(*!
<summary>Advances the cursor to the next source position.</summary>
<description>
The source must be live, non-null and structurally unchanged during traversal. TRUE identifies a current
entry. The index advances only while below source Length and stops at the end position. Repeated exhausted
calls return FALSE without incrementing the index; reading Current yields an empty descriptor. Reset allows
traversal from the beginning again. No snapshot or mutation detection is provided. Descendants cannot override
this cursor operation; advancement, reset and borrowed current views use the same cursor state.
Missing source raises DataMemberNotSpecifiedException before source access or cursor advancement.
</description>
*)
{attribute "object_name" := "MoveNext"}
METHOD FINAL MoveNext : BOOL
requireSource();

IF _CurrentIndex < _List.Length THEN
	_CurrentIndex := _CurrentIndex + 1;
END_IF

MoveNext := _CurrentIndex < _List.Length;
END_METHOD

(*!
<summary>Provides the library namespace for diagnostics.</summary>
<description>
Borrowed read-only reference to compiler-initialized metadata; no ownership transfer.
</description>
*)
{attribute 'monitoring' := 'call'}
PROPERTY NamespaceName : REFERENCE TO STRING
GET
NamespaceName REF= CurrentNamespace.Name;
END_GET
END_PROPERTY

(*!
<summary>Places the cursor before the first source entry.</summary>
<description>
The next MoveNext starts at zero. Does not modify the source or release payload; reading Current now yields an
empty descriptor. Descendants cannot override this cursor operation; advancement, reset and borrowed current
views use the same cursor state.
</description>
*)
{attribute "object_name" := "Reset"}
METHOD FINAL Reset
_CurrentIndex := -1;
END_METHOD

(*!
<summary>Reports the size of this function-block instance.</summary>
<description>
Measured in bytes; includes inline storage but excludes separately allocated buffers, payload and enumerators.
</description>
*)
{attribute 'monitoring' := 'call'}
PROPERTY SelfSize : ULINT
GET
SelfSize := XSIZEOF(THIS^);
END_GET
END_PROPERTY

(*!
<summary>Requires the configured source before traversal or current-value access.</summary>
<description>
A missing mandatory source is configuration failure, not an empty collection. Raises a framework diagnostic
outside lifecycle methods and before mutation; it does not validate arbitrary pointer lifetime.
</description>
*)
METHOD PRIVATE requireSource
IF _List = 0 THEN
	TOF_Core.Exceptions.ThrowDataMemberNotSpecified(
		sourceNamespaceName := NamespaceName,
		sourceClassName := ClassName,
		sourcePOUName := __POUNAME(),
		sourcePosition := __POSITION(),
		dataMemberName := 'list'
	);
END_IF
END_METHOD

END_FUNCTION_BLOCK

// ---- List/List.TcPOU
(*
SPDX-FileCopyrightText: © 2026 Oleksandr Tiutyk <trofimich@gmail.com>
SPDX-License-Identifier: MIT
License: https://opensource.org/license/mit
*)

(*!
<summary>Stores an ordered sequence of generic values with fixed or dynamic capacity.</summary>
<description>
CreateEnumerator allocates an independent cursor owned by its caller. The collection must remain alive while
that cursor is used. Dynamic growth preserves the existing buffer on allocation failure and invokes the
terminal allocation-failure mechanism. Sort uses GENERIC_VALUE.CompareTo unless an explicit borrowed comparer
is supplied; descriptors preserve OBJECT and USER_DEFINED categories. Successful insertion transfers disposal
responsibility for owned payload; borrowed payload must remain alive while stored. The caller-side descriptor
copy is not reset and must not be released again after transfer. Independent owning aliases and overlapping
owned allocations are unsupported. Entries retain order and duplicates. Same-allocation replacement preserves
ownership without releasing retained storage. Get, FindSingle and enumerators only borrow payload.
ContainsGeneric defaults to releasing its query. Validators are borrowed for the collection lifetime. No
locking or mutation-version checks are implemented; callbacks that mutate the collection can invalidate
in-progress operations. Generic lookup with requested query release also attempts cleanup on lookup failure
before propagating the captured exception; terminal OOM takes precedence.
Instances cannot be assigned by value: copying backing pointers or disposal responsibility would create
unsafe aliases. Interface references still borrow this instance; copying an interface does not clone storage.
</description>
*)

{attribute 'no_explicit_call' := 'do not call this function block directly'}
FUNCTION_BLOCK List 
VAR_GENERIC CONSTANT
 	{attribute 'hide'} 
	//! <summary>Inline capacity; zero selects dynamic backing storage.</summary>
	_StaticCapacity : TOF_Core.DINT_LENGTH := 0;
END_VAR
EXTENDS TOF_Core.Object IMPLEMENTS IList
VAR_INPUT
	//! <summary>Number of slots added when dynamic storage is full; must be positive when growth is required.</summary>
	DefaultDynamicAllocationElementCount : BYTE := 10;	
END_VAR
VAR_STAT
	//! <summary>Class name shared by all instances of this function block.</summary>
	{attribute 'hide'} 
	_ClassName : STRING := __POUNAME();
END_VAR
VAR
	{attribute 'hide'} 
	_ValueValidator : TOF_Core.IGenericValueValidator;

	{attribute 'hide'} 
	_Array : POINTER TO TOF_Core.GENERIC_VALUE;
	{attribute 'hide'} 
	_StaticArray : ARRAY [0.._StaticCapacity - 1] OF TOF_Core.GENERIC_VALUE;
	
	{attribute 'hide'} 
	_DynamicCapacity : TOF_Core.DINT_LENGTH;
	{attribute 'hide'} 
	_Length : TOF_Core.DINT_LENGTH;
END_VAR

(*!
<summary>Grows the dynamic element buffer while preserving existing values.</summary>
<description>
Static instances return without allocation. A positive increment must fit DINT capacity and the UDINT
allocation-byte limit; invalid ranges raise ArgumentOutOfRangeException before storage changes. A null
allocation invokes the terminal allocation-failure mechanism before copying or deleting the old buffer.
Existing descriptors are moved without cloning payload; incoming ownership is not accepted by this helper.
Descendants cannot override this storage operation; capacity, indexing and disposal remain governed by this
collection implementation.
</description>
*)
METHOD PROTECTED FINAL AllocateMemory 
VAR_INPUT
	elementCount : TOF_Core.DINT_LENGTH;
END_VAR
VAR CONSTANT
	//! <summary>Bytes per capacity slot, including descriptor storage and any hash-index arrays.</summary>
	ENTRY_ALLOCATION_SIZE : ULINT := XSIZEOF(TOF_Core.GENERIC_VALUE);
END_VAR
VAR
	newMemory : POINTER TO TOF_Core.GENERIC_VALUE;
	newCapacity : ULINT;

END_VAR
IF NOT Dynamic THEN
	RETURN;
END_IF

IF elementCount <= TOF_Core.SignedInt32.ZERO THEN
	TOF_Core.Exceptions.ThrowArgumentOutOfRange(
		sourceNamespaceName := NamespaceName,
		sourceClassName := ClassName,
		sourcePOUName := __POUNAME(),
		sourcePosition := __POSITION(),
		argumentName := 'elementCount',
		argumentValue := elementCount
	);
END_IF

newCapacity := TO_ULINT(_DynamicCapacity) + TO_ULINT(elementCount);

IF newCapacity > TO_ULINT(TOF_Core.SignedInt32.MAX_VALUE)
	OR_ELSE newCapacity > TO_ULINT(TOF_Core.UnsignedInt32.MAX_VALUE) / ENTRY_ALLOCATION_SIZE
THEN
	TOF_Core.Exceptions.ThrowArgumentOutOfRange(
		sourceNamespaceName := NamespaceName,
		sourceClassName := ClassName,
		sourcePOUName := __POUNAME(),
		sourcePosition := __POSITION(),
		argumentName := 'capacity',
		argumentValue := newCapacity
	);
END_IF

newMemory := __NEW(BYTE, TO_UDINT(ENTRY_ALLOCATION_SIZE * newCapacity));

IF newMemory = 0 THEN
	TOF_Core.DynamicMemoryManager.RaiseAllocationFailure();
END_IF

IF _Length > TOF_Core.SignedInt32.ZERO THEN
	Tc2_System.MEMCPY(destAddr := newMemory, srcAddr := _Array, n := TO_UDINT(ENTRY_ALLOCATION_SIZE * TO_ULINT(_Length)));
END_IF

IF _Array <> 0 THEN
	__DELETE(_Array);
END_IF

_DynamicCapacity := TO_DINT(newCapacity);
_Array := newMemory;
END_METHOD

(*!
<summary>Copies a value and appends the owned descriptor.</summary>
<description>
Borrows the original during the call. isObject = TRUE requires a live Object FB instance implementing
ICloneable; other data is copied as bytes without recursively cloning references. A prepared copy is released
if insertion fails before acceptance; exceptions propagate. Engine-managed exception objects are unsupported.
index is meaningful only on success. Descendants cannot override this storage operation; capacity, indexing
and disposal remain governed by this collection implementation.
The original failure is captured before cleanup so nested cleanup handling cannot replace its payload.
A static native wrapper is cloned before cleanup; failure to capture still attempts prepared-copy disposal.
Terminal allocation failure takes precedence and no exception clone is allocated after its latch is set.
</description>
*)
METHOD FINAL AppendCopy : IList
VAR_INPUT
	value : ANY;
	isObject : BOOL := FALSE;
END_VAR
VAR_OUTPUT
	index : TOF_Core.DINT_INDEX;
END_VAR
VAR
	exceptionCode : __SYSTEM.ExceptionCode;
	caughtException : TOF_Core.IException;
	genericValue : TOF_Core.GENERIC_VALUE;
END_VAR

genericValue := TOF_Core.GenericValueFactory.FromAnyType(
		value := value,
		isObject := isObject,
		memoryManagementBehavior := TOF_Core.GENERIC_MEMORY_MANAGEMENT_BEHAVIOR.CLONE_ORIGINAL_VALUE_AND_OWNS_MEMORY
	);

__TRY
	AppendCopy := AppendGeneric(value := genericValue, index => index);
__CATCH(exceptionCode)
	caughtException := TOF_Core.ExceptionManager.GetLastException(
		exceptionCode := exceptionCode,
		catchPointNamespaceName := NamespaceName,
		catchPointPOUName := __POUNAME(),
		catchPointPosition := __POSITION()
	);
__ENDTRY

IF caughtException <> 0 THEN
	__TRY
		TOF_Core.DynamicMemoryManager.RaiseIfAllocationFailed();

		IF NOT caughtException.IsDynamicInstance THEN
			__QUERYINTERFACE(caughtException.Clone(), caughtException);
		END_IF
	__CATCH(exceptionCode)
		genericValue.Release();

		TOF_Core.ExceptionManager.ReThrowLastException(
			exceptionCode := exceptionCode,
			catchPointNamespaceName := NamespaceName,
			catchPointPOUName := __POUNAME(),
			catchPointPosition := __POSITION()
		);
	__ENDTRY

	genericValue.Release();

	TOF_Core.ExceptionManager.Throw(exception := caughtException);
END_IF
END_METHOD

(*!
<summary>Appends a descriptor to the list.</summary>
<description>
Successful insertion transfers disposal responsibility for owned payload; borrowed payload must remain alive
while stored. The caller-side descriptor copy is not reset and must not be released again after transfer.
Independent owning aliases and overlapping owned allocations are unsupported. Delegates to InsertGeneric;
index is meaningful only on success. Descendants cannot override this storage operation; capacity, indexing
and disposal remain governed by this collection implementation.
</description>
*)
METHOD FINAL AppendGeneric : IList
VAR_INPUT
	value : TOF_Core.GENERIC_VALUE;
END_VAR
VAR_OUTPUT
	index : TOF_Core.DINT_INDEX;
END_VAR
index := _Length;

AppendGeneric := InsertGeneric(index := index, value := value);
END_METHOD

(*!
<summary>Reports the currently allocated number of slots.</summary>
<description>
Units are bytes for ByteList and entries for other collections. Static capacity is fixed; dynamic capacity can
change on growth or clearing. This is not a guarantee that the next allocation succeeds.
</description>
*)
{attribute 'monitoring' := 'call'}
PROPERTY FINAL Capacity : TOF_Core.DINT_LENGTH
GET
Capacity := SEL(_StaticCapacity = 0, _StaticCapacity, _DynamicCapacity);
END_GET
END_PROPERTY

(*!
<summary>Borrows the concrete collection class name without transferring storage ownership.</summary>
*)
{attribute 'monitoring' := 'call'}
PROPERTY ClassName : REFERENCE TO STRING
GET
ClassName REF= _ClassName;
END_GET
END_PROPERTY

(*!
<summary>Removes all entries and releases dynamic backing storage.</summary>
<description>
Owned payload is released best effort through GENERIC_VALUE.Release; borrowed storage is not freed. Static
capacity and the borrowed validator are retained. Dynamic capacity becomes zero. Returns this collection and
invalidates positions and views. Cleanup callbacks must not reenter mutation. Descendants cannot override this
storage operation; capacity, indexing and disposal remain governed by this collection implementation.
</description>
*)
METHOD FINAL Clear : IList
VAR
	i : DINT;
END_VAR
Clear := THIS^;

FOR i := 0 TO _Length - 1 DO
	_Array[i].Release();						
END_FOR	

_Length := 0;
_DynamicCapacity := 0;

IF _Array <> 0 AND_THEN Dynamic THEN
	__DELETE(_Array);	
END_IF
END_METHOD

(*!
<summary>Searches for a value using default generic equality.</summary>
<description>
Borrows the ANY argument during a linear search without cloning or releasing it. isObject = TRUE means a live
Object FB instance, not a pointer or interface variable. Equality exceptions propagate; callbacks that mutate
the collection can invalidate traversal. Descendants cannot override this storage operation; capacity,
indexing and disposal remain governed by this collection implementation.
</description>
*)
METHOD FINAL Contains : BOOL
VAR_INPUT
	value : ANY;
	isObject : BOOL := FALSE;
END_VAR
VAR
	genericValue : TOF_Core.GENERIC_VALUE;
	i : TOF_Core.DINT_INDEX;
END_VAR

genericValue := TOF_Core.GenericValueFactory.FromAnyType(
		value := value,
		isObject := isObject,
		memoryManagementBehavior := TOF_Core.GENERIC_MEMORY_MANAGEMENT_BEHAVIOR.STORE_ORIGINAL_REFERENCE_AND_NOT_OWNS_MEMORY
	);

FOR i := 0 TO _Length - 1 DO
	IF _Array[i].Equals(otherValue := genericValue) THEN
		Contains := TRUE;
		RETURN;
	END_IF
END_FOR
END_METHOD

(*!
<summary>Searches for an equal generic value and optionally releases the query.</summary>
<description>
Uses GENERIC_VALUE.Equals in a linear search. releaseValue defaults to TRUE: after a completed search, Release
is called on the local query copy, including on a miss. Caller-side aliases are not reset. The query must not
own storage retained by the collection. Requested release is attempted after both successful lookup and lookup
failure. Before cleanup, the original framework exception is retained and a borrowed static system exception
is cloned to preserve its code, catch point and timestamps across cleanup callbacks. The captured exception is
then propagated through ExceptionManager.Throw in the current cyclic task; native errors use the framework
SystemException representation. If capturing the system exception fails with terminal OOM, query cleanup is
still attempted and terminal OOM takes precedence. Terminal allocation state is never cleared. Release is best
effort and does not prove successful deallocation. Cleanup callbacks must not reenter collection mutation.
Descendants cannot override this storage operation; capacity, indexing and disposal remain governed by this
collection implementation.
</description>
*)
METHOD FINAL ContainsGeneric : BOOL
VAR_INPUT
	value : TOF_Core.GENERIC_VALUE;
	releaseValue : BOOL := TRUE;
END_VAR
VAR
	exceptionCode : __SYSTEM.ExceptionCode;
	caughtException : TOF_Core.IException;

	i : DINT;
END_VAR
__TRY
	FOR i := 0 TO _Length - 1 DO
		IF _Array[i].Equals(otherValue := value) THEN
			ContainsGeneric := TRUE;
			EXIT;
		END_IF
	END_FOR
__CATCH(exceptionCode)
	caughtException := TOF_Core.ExceptionManager.GetLastException(
		exceptionCode := exceptionCode,
		catchPointNamespaceName := NamespaceName,
		catchPointPOUName := __POUNAME(),
		catchPointPosition := __POSITION()
	);
__ENDTRY

IF releaseValue THEN
	IF caughtException <> 0 AND_THEN NOT caughtException.IsDynamicInstance THEN
		__TRY
			TOF_Core.DynamicMemoryManager.RaiseIfAllocationFailed();
			__QUERYINTERFACE(caughtException.Clone(), caughtException);
		__CATCH(exceptionCode)
			value.Release();

			TOF_Core.ExceptionManager.ReThrowLastException(
				exceptionCode := exceptionCode,
				catchPointNamespaceName := NamespaceName,
				catchPointPOUName := __POUNAME(),
				catchPointPosition := __POSITION()
			);
		__ENDTRY
	END_IF

	value.Release();
END_IF

IF caughtException <> 0 THEN
	TOF_Core.ExceptionManager.Throw(exception := caughtException);
END_IF
END_METHOD

(*!
<summary>Creates an independent enumerator owned by the caller.</summary>
<description>
The caller must explicitly release the enumerator and keep this collection alive while using it. Allocation
failure invokes DynamicMemoryManager.RaiseAllocationFailure without a heap exception; it is terminal and is
not returned as a recoverable null result.
</description>
*)
METHOD CreateEnumerator : TOF_Core.IEnumerator
VAR
	enumerator : POINTER TO ListEnumerator;
END_VAR
enumerator := __NEW(ListEnumerator(list := THIS^));

IF enumerator = 0 THEN
	TOF_Core.DynamicMemoryManager.RaiseAllocationFailure();
END_IF

CreateEnumerator := enumerator^;
END_METHOD

(*!
<summary>Reports whether storage can grow dynamically.</summary>
<description>
Static capacity zero selects dynamic storage. Dynamic collections can still fail to allocate.
</description>
*)
{attribute 'monitoring' := 'call'}
PROPERTY FINAL Dynamic : BOOL
GET
Dynamic := _StaticCapacity = 0;
END_GET
END_PROPERTY

(*!
<summary>Reports whether the collection has no entries.</summary>
<description>
Reflects Length; not a check of payload lifetime or memory health.
</description>
*)
{attribute 'monitoring' := 'call'}
PROPERTY FINAL Empty : BOOL
GET
Empty := _Length <= 0;
END_GET
END_PROPERTY

(*!
<summary>Releases owned payload and backing storage during destruction.</summary>
<description>
Calls Clear; lifecycle methods and payload cleanup callbacks must not raise exceptions or reenter mutation.
Payload release is best effort, not proof of successful destruction. No separate copy-code ownership handoff
is implemented.
</description>
*)

METHOD FB_exit : BOOL
VAR_INPUT
	bInCopyCode : BOOL; 
END_VAR
Clear();
END_METHOD

(*!
<summary>Binds the optional validator and inline storage during initialization.</summary>
<description>
The validator is borrowed and must remain alive while used; it is not invoked here. Static storage is bound
without allocation. Lifecycle methods must not raise exceptions. No explicit online-change relocation repair
is implemented.
</description>
*)
METHOD FB_init : BOOL
VAR_INPUT
	bInitRetains : BOOL; // TRUE: the retain variables are initialized (reset warm / reset cold)
	bInCopyCode : BOOL; // TRUE: the instance will be copied to the copy code afterward (online change)
	valueValidator : TOF_Core.IGenericValueValidator;
END_VAR
_ValueValidator := valueValidator;

IF NOT Dynamic THEN
	_Array := ADR(_StaticArray); 
END_IF
END_METHOD

(*!
<summary>Finds a predicate match in the requested traversal direction.</summary>
<description>
skip counts matches, not visited entries. A null predicate or no match returns FALSE; outputs are meaningful
only on TRUE. The result is borrowed even if IsMemoryOwner is TRUE. Predicate input uses AsAnyType without
preserving the explicit generic OBJECT category. Predicate exceptions propagate; callbacks must not mutate the
traversed collection. Descendants cannot override this storage operation; capacity, indexing and disposal
remain governed by this collection implementation.
</description>
*)
METHOD FINAL FindSingle : BOOL
VAR_INPUT
	predicate : TOF_Core.IPredicate;
	skip : UDINT := 0;
	searchDirection : TOF_Core.SEARCH_DIRECTION := TOF_Core.SEARCH_DIRECTION.FROM_BEGINNING;
END_VAR
VAR_OUTPUT
	value : TOF_Core.GENERIC_VALUE;
	index : TOF_Core.DINT_INDEX;
END_VAR
VAR
	startSearchIndex : DINT;
	maxSearchIndex : DINT;
	indexStep : DINT;
	
	i : DINT;
	
	currentValue : __SYSTEM.AnyType;

	skippedMatchCount : UDINT := 0;
END_VAR
index := 0;
	
IF TO_DINT(skip) >= _Length OR_ELSE predicate = 0 THEN
	RETURN;
END_IF

startSearchIndex := SEL(searchDirection = TOF_Core.SEARCH_DIRECTION.FROM_BEGINNING, _Length - 1, 0);
maxSearchIndex := SEL(searchDirection = TOF_Core.SEARCH_DIRECTION.FROM_BEGINNING, 0, _Length - 1);
indexStep := SEL(searchDirection = TOF_Core.SEARCH_DIRECTION.FROM_BEGINNING, -1, 1);

FOR i := startSearchIndex TO maxSearchIndex BY indexStep DO
	currentValue := _Array[i].AsAnyType();
	
	IF predicate.Check(valueToCompare := currentValue) THEN
		IF skip = skippedMatchCount THEN
			value := _Array[i];
			index := i;
			FindSingle := TRUE;
			RETURN;
		ELSE
			skippedMatchCount := skippedMatchCount + 1;
		END_IF
	END_IF
END_FOR
END_METHOD

(*!
<summary>Reports whether fixed-capacity storage has no free slot.</summary>
<description>
Dynamic collections report FALSE even when Length equals Capacity. This does not guarantee available heap
memory.
</description>
*)
{attribute 'monitoring' := 'call'}
PROPERTY FINAL Full : BOOL
GET
Full := _StaticCapacity <> 0 AND_THEN _Length >= _StaticCapacity;
END_GET
END_PROPERTY

(*!
<summary>Borrows the descriptor at a zero-based list position.</summary>
<description>
An out-of-range index raises an exception. Returned descriptors and payload are borrowed, not clones. Do not
modify descriptor metadata or release payload through this view, even when IsMemoryOwner is TRUE. Keep the
source and borrowed storage alive; mutation or destruction can invalidate the view. Descendants cannot
override this storage operation; capacity, indexing and disposal remain governed by this collection
implementation.
</description>
*)
METHOD FINAL Get : REFERENCE TO TOF_Core.GENERIC_VALUE
VAR_INPUT
	index : TOF_Core.DINT_INDEX;
END_VAR
IF index < 0 OR_ELSE index >= _Length THEN
	TOF_Core.Exceptions.ThrowArgumentOutOfRange(
		sourceNamespaceName := NamespaceName,
		sourceClassName := ClassName,
		sourcePOUName := __POUNAME(),
		sourcePosition := __POSITION(),
		argumentName := 'index',
		argumentValue := index
	);
END_IF

Get REF= _Array[index];
END_METHOD

(*!
<summary>Copies a value and inserts it at the requested position.</summary>
<description>
Borrows the original during the call. isObject = TRUE requires a live Object FB instance implementing
ICloneable; other data is copied as bytes without recursively cloning references. A prepared copy is released
if insertion fails before acceptance; exceptions propagate. Engine-managed exception objects are unsupported.
The position may range from zero through Length inclusive. Descendants cannot override this storage operation;
capacity, indexing and disposal remain governed by this collection implementation.
The original failure is captured before cleanup so nested cleanup handling cannot replace its payload.
A static native wrapper is cloned before cleanup; failure to capture still attempts prepared-copy disposal.
Terminal allocation failure takes precedence and no exception clone is allocated after its latch is set.
</description>
*)
METHOD FINAL InsertCopy : IList
VAR_INPUT
	index : TOF_Core.DINT_INDEX;
	value : ANY;
	isObject : BOOL := FALSE;
END_VAR
VAR
	exceptionCode : __SYSTEM.ExceptionCode;
	caughtException : TOF_Core.IException;
	genericValue : TOF_Core.GENERIC_VALUE;
END_VAR

genericValue := TOF_Core.GenericValueFactory.FromAnyType(
		value := value,
		isObject := isObject,
		memoryManagementBehavior := TOF_Core.GENERIC_MEMORY_MANAGEMENT_BEHAVIOR.CLONE_ORIGINAL_VALUE_AND_OWNS_MEMORY
	);

__TRY
	InsertCopy := InsertGeneric(index := index, value := genericValue);
__CATCH(exceptionCode)
	caughtException := TOF_Core.ExceptionManager.GetLastException(
		exceptionCode := exceptionCode,
		catchPointNamespaceName := NamespaceName,
		catchPointPOUName := __POUNAME(),
		catchPointPosition := __POSITION()
	);
__ENDTRY

IF caughtException <> 0 THEN
	__TRY
		TOF_Core.DynamicMemoryManager.RaiseIfAllocationFailed();

		IF NOT caughtException.IsDynamicInstance THEN
			__QUERYINTERFACE(caughtException.Clone(), caughtException);
		END_IF
	__CATCH(exceptionCode)
		genericValue.Release();

		TOF_Core.ExceptionManager.ReThrowLastException(
			exceptionCode := exceptionCode,
			catchPointNamespaceName := NamespaceName,
			catchPointPOUName := __POUNAME(),
			catchPointPosition := __POSITION()
		);
	__ENDTRY

	genericValue.Release();

	TOF_Core.ExceptionManager.Throw(exception := caughtException);
END_IF
END_METHOD

(*!
<summary>Inserts a descriptor and shifts subsequent entries to the right.</summary>
<description>
Successful insertion transfers disposal responsibility for owned payload; borrowed payload must remain alive
while stored. The caller-side descriptor copy is not reset and must not be released again after transfer.
Independent owning aliases and overlapping owned allocations are unsupported. index may range from zero
through Length inclusive. Invalid indices and full static storage raise exceptions. Validation precedes
insertion. Dynamic growth rejects nonpositive increments and unrepresentable capacity or allocation sizes
before insertion. Descendants cannot override this storage operation; capacity, indexing and disposal remain
governed by this collection implementation.
</description>
*)
METHOD FINAL InsertGeneric : IList
VAR_INPUT
	index : TOF_Core.DINT_INDEX;
	value : TOF_Core.GENERIC_VALUE;	
END_VAR
VAR
	
	i : DINT;
END_VAR
IF index < 0 OR_ELSE index > _Length THEN
	TOF_Core.Exceptions.ThrowArgumentOutOfRange(
		sourceNamespaceName := NamespaceName,
		sourceClassName := ClassName,
		sourcePOUName := __POUNAME(),
		sourcePosition := __POSITION(),
		argumentName := 'index',
		argumentValue := index
	);
END_IF

IF _ValueValidator <> 0 THEN
	_ValueValidator.Validate(validatedObjectName := GetName(), valueToValidate := value);
END_IF

InsertGeneric := THIS^;

IF _Length >= Capacity THEN
	IF Dynamic THEN
		AllocateMemory(elementCount := DefaultDynamicAllocationElementCount);
	ELSE
		TOF_Core.Exceptions.ThrowStaticCollectionFull(
			sourceNamespaceName := NamespaceName,
			sourceClassName := ClassName,
			sourcePOUName := __POUNAME(),
			sourcePosition := __POSITION(),
			collectionName := GetName(),
			capacity := TO_UDINT(Capacity)
		);
	END_IF
END_IF

_Length := _Length + 1;

i := _Length - 1;

WHILE i > index DO
	_Array[i] := _Array[i - 1];	
	i := i - 1;
END_WHILE

_Array[i] := value;
END_METHOD

(*!
<summary>Reports the number of stored entries.</summary>
<description>
Units are bytes for ByteList and entries for other collections. Existing positions range from zero through
Length minus one.
</description>
*)
{attribute 'monitoring' := 'call'}
PROPERTY FINAL Length : TOF_Core.DINT_LENGTH
GET
Length := _Length;
END_GET
END_PROPERTY

(*!
<summary>Provides the library namespace for diagnostics.</summary>
<description>
Borrowed read-only reference to compiler-initialized metadata; no ownership transfer.
</description>
*)
{attribute 'monitoring' := 'call'}
PROPERTY NamespaceName : REFERENCE TO STRING
GET
NamespaceName REF= CurrentNamespace.Name;
END_GET
END_PROPERTY

(*!
<summary>Removes an existing list entry and compacts subsequent entries.</summary>
<description>
Invalid indices raise an exception. Owned payload is released best effort through GENERIC_VALUE.Release;
borrowed payload is not freed. Returns this list. Positions and descriptor references may change; cleanup
callbacks must not reenter mutation. Descendants cannot override this storage operation; capacity, indexing
and disposal remain governed by this collection implementation.
</description>
*)
METHOD FINAL RemoveAt : IList
VAR_INPUT
	index : TOF_Core.DINT_INDEX;
END_VAR
IF index < 0 OR_ELSE index >= _Length THEN
	TOF_Core.Exceptions.ThrowArgumentOutOfRange(
		sourceNamespaceName := NamespaceName,
		sourceClassName := ClassName,
		sourcePOUName := __POUNAME(),
		sourcePosition := __POSITION(),
		argumentName := 'index',
		argumentValue := index
	);
END_IF

RemoveAt := THIS^;

_Array[index].Release();			

IF index < _Length - 1 THEN
	Tc2_System.MEMMOVE(
		destAddr := ADR(_Array[index]),
		srcAddr := ADR(_Array[index + 1]),
		n := TO_UDINT(SIZEOF(TOF_Core.GENERIC_VALUE) * (_Length - index - 1))
	);
END_IF

_Array[_Length - 1].Reset();	

_Length := _Length - 1;
END_METHOD

(*!
<summary>Removes the first list entry equal to a borrowed query.</summary>
<description>
Uses default GENERIC_VALUE equality; isObject = TRUE requires a live Object FB instance. Reports removed on a
successful match and returns this list. Owned stored payload is released; the query is not adopted or
separately released. Equality exceptions propagate. Descendants cannot override this storage operation;
capacity, indexing and disposal remain governed by this collection implementation.
</description>
*)
METHOD FINAL RemoveFirst : IList
VAR_INPUT
	value : ANY;
	isObject : BOOL := FALSE;
END_VAR
VAR_OUTPUT
	removed : BOOL;
END_VAR
VAR
	genericValue : TOF_Core.GENERIC_VALUE;
	i : TOF_Core.DINT_INDEX;
END_VAR
RemoveFirst := THIS^;

IF _Length > 0 THEN
	genericValue := TOF_Core.GenericValueFactory.FromAnyType(
		value := value,
		isObject := isObject,
		memoryManagementBehavior := TOF_Core.GENERIC_MEMORY_MANAGEMENT_BEHAVIOR.STORE_ORIGINAL_REFERENCE_AND_NOT_OWNS_MEMORY
	);
	
	FOR i := 0 TO _Length - 1 DO
		IF _Array[i].Equals(otherValue := genericValue) THEN
			RemoveAt(index := i);
			removed := TRUE;
			RETURN;
		END_IF
	END_FOR
END_IF
END_METHOD

(*!
<summary>Removes predicate matches while traversing from the end.</summary>
<description>
skip counts matches from the end. A null predicate or maxRemoved = 0 performs no removal. Removes at most
maxRemoved matching entries after skipping the requested matches. Stops immediately after reaching the limit,
without invoking the predicate for remaining entries. Predicate exceptions propagate after any completed
removals, without rollback. removedCount counts completed removals. Callbacks must not mutate the traversed
collection. Descendants cannot override this storage operation; capacity, indexing and disposal remain
governed by this collection implementation.
</description>
*)
METHOD FINAL RemoveMatched : IList
VAR_INPUT
	predicate : TOF_Core.IPredicate;
	skip : UDINT := 0;
	maxRemoved : UDINT := TOF_Core.UnsignedInt32.MAX_VALUE;
END_VAR
VAR_OUTPUT
	removedCount : DINT;
END_VAR
VAR
	i : DINT;

	currentValue : __SYSTEM.AnyType;

	skippedMatchCount : UDINT := 0;
END_VAR
RemoveMatched := THIS^;

IF TO_DINT(skip) >= _Length OR_ELSE predicate = 0 OR_ELSE maxRemoved = TOF_Core.UnsignedInt32.MIN_VALUE THEN
	RETURN;
END_IF

FOR i := _Length - 1 TO 0 BY -1 DO
	currentValue := _Array[i].AsAnyType();
	
	IF predicate.Check(valueToCompare := currentValue) THEN
		IF skip <= skippedMatchCount THEN
			RemoveAt(index := i);
			removedCount := removedCount + 1;

			IF TO_UDINT(removedCount) >= maxRemoved THEN
				EXIT;
			END_IF
		ELSE
			skippedMatchCount := skippedMatchCount + 1;
		END_IF
	END_IF
END_FOR
END_METHOD

(*!
<summary>Restores the heap order below a root within the active sort range.</summary>
<description>
Requires valid indices and the same ordering selection used by Sort. A null comparer selects
GENERIC_VALUE.CompareTo; an explicit comparer takes precedence. Uses typed entry addresses and swaps
complete descriptors in place. Comparison exceptions propagate without rolling back completed swaps.
</description>
*)
METHOD PRIVATE restoreHeapFrom
VAR_INPUT
	rootIndex : DINT;
	heapSize : DINT;
	comparer : TOF_Core.IComparer;
	direction : TOF_Core.SORT_DIRECTION;
END_VAR
VAR
	currentIndex : DINT;
	childIndex : DINT;
	selectedIndex : DINT;

	comparisonResult : TOF_Core.COMPARISON_RESULT;

	value1, value2 : POINTER TO TOF_Core.GENERIC_VALUE;
END_VAR
currentIndex := rootIndex;

WHILE (currentIndex * 2 + 1) < heapSize DO
	childIndex := currentIndex * 2 + 1;
	selectedIndex := currentIndex;

	value1 := ADR(_Array[selectedIndex]);
	value2 := ADR(_Array[childIndex]);

	IF comparer = 0 THEN
		comparisonResult := value1^.CompareTo(otherValue := value2^);
	ELSE
		comparisonResult := comparer.Compare(first := value1^, second := value2^);
	END_IF

	IF direction = TOF_Core.SORT_DIRECTION.ASCENDING THEN
		IF comparisonResult = TOF_Core.COMPARISON_RESULT.FIRST_LESS_THAN_SECOND THEN
			selectedIndex := childIndex;
		END_IF
	ELSE
		IF comparisonResult = TOF_Core.COMPARISON_RESULT.FIRST_GREATER_THAN_SECOND THEN
			selectedIndex := childIndex;
		END_IF
	END_IF

	IF (childIndex + 1) < heapSize THEN
		value1 := ADR(_Array[selectedIndex]);
		value2 := ADR(_Array[childIndex + 1]);

		IF comparer = 0 THEN
			comparisonResult := value1^.CompareTo(otherValue := value2^);
		ELSE
			comparisonResult := comparer.Compare(first := value1^, second := value2^);
		END_IF

		IF direction = TOF_Core.SORT_DIRECTION.ASCENDING THEN
			IF comparisonResult = TOF_Core.COMPARISON_RESULT.FIRST_LESS_THAN_SECOND THEN
				selectedIndex := childIndex + 1;
			END_IF
		ELSE
			IF comparisonResult = TOF_Core.COMPARISON_RESULT.FIRST_GREATER_THAN_SECOND THEN
				selectedIndex := childIndex + 1;
			END_IF
		END_IF
	END_IF

	IF selectedIndex = currentIndex THEN
		RETURN;
	END_IF

	Swap(index1 := currentIndex, index2 := selectedIndex);
	
	currentIndex := selectedIndex;
END_WHILE
END_METHOD

(*!
<summary>Reports the size of this function-block instance.</summary>
<description>
Measured in bytes; includes inline storage but excludes separately allocated buffers, payload and enumerators.
</description>
*)
{attribute 'monitoring' := 'call'}
PROPERTY SelfSize : ULINT
GET
SelfSize := XSIZEOF(THIS^);
END_GET
END_PROPERTY

(*!
<summary>Copies a value and stores it through SetGeneric.</summary>
<description>
Borrows the original during the call. isObject = TRUE requires a live Object FB instance implementing
ICloneable; other data is copied as bytes without recursively cloning references. A prepared copy is released
if insertion fails before acceptance; exceptions propagate. Engine-managed exception objects are unsupported.
Any index output is meaningful only on success. Descendants cannot override this storage operation; capacity,
indexing and disposal remain governed by this collection implementation.
The original failure is captured before cleanup so nested cleanup handling cannot replace its payload.
A static native wrapper is cloned before cleanup; failure to capture still attempts prepared-copy disposal.
Terminal allocation failure takes precedence and no exception clone is allocated after its latch is set.
</description>
*)
METHOD FINAL SetCopy : IList
VAR_INPUT
	index : TOF_Core.DINT_INDEX;
	value : ANY;
	isObject : BOOL := FALSE;
END_VAR
VAR
	exceptionCode : __SYSTEM.ExceptionCode;
	caughtException : TOF_Core.IException;
	genericValue : TOF_Core.GENERIC_VALUE;
END_VAR

genericValue := TOF_Core.GenericValueFactory.FromAnyType(
		value := value,
		isObject := isObject,
		memoryManagementBehavior := TOF_Core.GENERIC_MEMORY_MANAGEMENT_BEHAVIOR.CLONE_ORIGINAL_VALUE_AND_OWNS_MEMORY
	);

__TRY
	SetCopy := SetGeneric(index := index, value := genericValue);
__CATCH(exceptionCode)
	caughtException := TOF_Core.ExceptionManager.GetLastException(
		exceptionCode := exceptionCode,
		catchPointNamespaceName := NamespaceName,
		catchPointPOUName := __POUNAME(),
		catchPointPosition := __POSITION()
	);
__ENDTRY

IF caughtException <> 0 THEN
	__TRY
		TOF_Core.DynamicMemoryManager.RaiseIfAllocationFailed();

		IF NOT caughtException.IsDynamicInstance THEN
			__QUERYINTERFACE(caughtException.Clone(), caughtException);
		END_IF
	__CATCH(exceptionCode)
		genericValue.Release();

		TOF_Core.ExceptionManager.ReThrowLastException(
			exceptionCode := exceptionCode,
			catchPointNamespaceName := NamespaceName,
			catchPointPOUName := __POUNAME(),
			catchPointPosition := __POSITION()
		);
	__ENDTRY

	genericValue.Release();

	TOF_Core.ExceptionManager.Throw(exception := caughtException);
END_IF
END_METHOD

(*!
<summary>Replaces the descriptor at an existing list position.</summary>
<description>
Successful replacement transfers disposal responsibility for owned payload; borrowed payload must remain alive
while stored. The caller-side descriptor copy is not reset and must not be released again after transfer.
Invalid indices and rejected validation raise exceptions before replacement. Reusing the same allocation
preserves existing ownership or accepts incoming ownership without releasing that allocation. Aliases must
have compatible disposal semantics; independently owned aliases and overlapping owned ranges are unsupported.
A different displaced allocation is released best effort after installing the new descriptor. Cleanup
callbacks must not reenter collection mutation. Descendants cannot override this storage operation; capacity,
indexing and disposal remain governed by this collection implementation.
</description>
*)
METHOD FINAL SetGeneric : IList
VAR_INPUT
	index : TOF_Core.DINT_INDEX;
	value : TOF_Core.GENERIC_VALUE;	
END_VAR
VAR

	displacedValue : TOF_Core.GENERIC_VALUE;
END_VAR
IF index < TOF_Core.SignedInt32.ZERO OR_ELSE index >= _Length THEN
	TOF_Core.Exceptions.ThrowArgumentOutOfRange(
		sourceNamespaceName := NamespaceName,
		sourceClassName := ClassName,
		sourcePOUName := __POUNAME(),
		sourcePosition := __POSITION(),
		argumentName := 'index',
		argumentValue := index
	);
END_IF

IF _ValueValidator <> 0 THEN
	_ValueValidator.Validate(validatedObjectName := GetName(), valueToValidate := value);
END_IF

SetGeneric := THIS^;

displacedValue := _Array[index];

IF displacedValue.Address = value.Address THEN
	IF displacedValue.IsMemoryOwner AND_THEN NOT value.IsMemoryOwner THEN
		value := TOF_Core.GenericValueFactory.FromParts(
			genericTypeClass := value.TypeClass,
			address := value.Address,
			size := value.Size,
			memoryManagementBehavior := TOF_Core.GENERIC_MEMORY_MANAGEMENT_BEHAVIOR.STORE_ORIGINAL_REFERENCE_AND_OWNS_MEMORY
		);
	END_IF

	displacedValue.Reset();
END_IF

_Array[index] := value;
displacedValue.Release();
END_METHOD

(*!
<summary>Reorders entries in place using the supplied generic-value ordering strategy.</summary>
<description>
A null or omitted comparer selects GENERIC_VALUE.CompareTo for each pair. An explicit comparer takes
precedence and must provide a consistent order for the stored representations. Payload and comparer are
borrowed. The default order supports Core numeric, text, temporal and OBJECT comparison rules; incompatible
pairs raise GenericConversionNotSupportedException and OBJECT values require IComparable. Empty and singleton
lists return without invoking comparisons. Callbacks must not modify operands or the collection. Exceptions
propagate without rolling back completed swaps; every descriptor and its ownership remain in the list.
Returns this list. Descendants cannot override the storage operation.
</description>
*)
//!<param name="comparer">Optional borrowed ordering strategy; zero selects GENERIC_VALUE.CompareTo.</param>
//!<param name="direction">Requested ordering direction.</param>
METHOD FINAL Sort : IList
VAR_INPUT
	comparer : TOF_Core.IComparer := 0;
	direction : TOF_Core.SORT_DIRECTION := TOF_Core.SORT_DIRECTION.ASCENDING;
END_VAR
VAR CONSTANT
	//! <summary>Largest entry count using insertion sort; larger lists use in-place heap sort.</summary>
	SMALL_LIST_SORT_LIMIT : DINT := 16;
END_VAR
VAR

	i : DINT;
	j : DINT;
	startIndex : DINT;
	endIndex : DINT;

	comparisonResult : TOF_Core.COMPARISON_RESULT;

	value1, value2 : TOF_Core.GENERIC_VALUE;
END_VAR
Sort := THIS^;

IF _Length <= 1 THEN
	RETURN;
END_IF

// Insertion sort is faster for small lists, otherwise use heap sort
IF _Length <= SMALL_LIST_SORT_LIMIT THEN
	FOR i := 1 TO _Length - 1 DO
		j := i;

		WHILE j > 0 DO
			value1 := _Array[j - 1];
			value2 := _Array[j];

			IF comparer = 0 THEN
				comparisonResult := value1.CompareTo(otherValue := value2);
			ELSE
				comparisonResult := comparer.Compare(first := value1, second := value2);
			END_IF

			IF direction = TOF_Core.SORT_DIRECTION.ASCENDING THEN
				IF comparisonResult <> TOF_Core.COMPARISON_RESULT.FIRST_GREATER_THAN_SECOND THEN
					EXIT;
				END_IF
			ELSE
				IF comparisonResult <> TOF_Core.COMPARISON_RESULT.FIRST_LESS_THAN_SECOND THEN
					EXIT;
				END_IF
			END_IF

			Swap(index1 := j - 1, index2 := j);
			
			j := j - 1;
		END_WHILE
	END_FOR

	RETURN;
END_IF

// Build heap
startIndex := (_Length / 2) - 1;

WHILE startIndex >= 0 DO
	restoreHeapFrom(rootIndex := startIndex, heapSize := _Length, comparer := comparer, direction := direction);
	
	startIndex := startIndex - 1;
END_WHILE

// Extract heap root into the final sorted position
endIndex := _Length - 1;

WHILE endIndex > 0 DO
	Swap(index1 := 0, index2 := endIndex);
	
	restoreHeapFrom(rootIndex := 0, heapSize := endIndex, comparer := comparer, direction := direction);
	
	endIndex := endIndex - 1;
END_WHILE
END_METHOD

(*!
<summary>Exchanges two positions without cloning or releasing payload.</summary>
<description>
Returns this list. Different indices must be valid or an exception is raised. Current implementation returns
immediately for equal indices without validating them. Payload ownership is preserved. Descendants cannot
override this storage operation; capacity, indexing and disposal remain governed by this collection
implementation.
</description>
*)
METHOD FINAL Swap : IList
VAR_INPUT
	index1 : TOF_Core.DINT_INDEX;
	index2 : TOF_Core.DINT_INDEX;
END_VAR
VAR
	tmp : TOF_Core.GENERIC_VALUE;
END_VAR
Swap := THIS^;

IF index1 = index2 THEN
	RETURN;
ELSIF index1 < 0 OR_ELSE index1 >= _Length THEN
	TOF_Core.Exceptions.ThrowArgumentOutOfRange(
		sourceNamespaceName := NamespaceName,
		sourceClassName := ClassName,
		sourcePOUName := __POUNAME(),
		sourcePosition := __POSITION(),
		argumentName := 'index1',
		argumentValue := index1
	);
ELSIF index2 < 0 OR_ELSE index2 >= _Length THEN
	TOF_Core.Exceptions.ThrowArgumentOutOfRange(
		sourceNamespaceName := NamespaceName,
		sourceClassName := ClassName,
		sourcePOUName := __POUNAME(),
		sourcePosition := __POSITION(),
		argumentName := 'index2',
		argumentValue := index2
	);
END_IF

tmp := _Array[index1];
_Array[index1] := _Array[index2];
_Array[index2] := tmp;
END_METHOD

(*!
<summary>Exposes the configured value validator.</summary>
<description>
Borrowed optional reference fixed at initialization. Zero means no validator. The collection does not own or
release it.
</description>
*)
{attribute 'monitoring' := 'call'}
PROPERTY FINAL ValueValidator : TOF_Core.IGenericValueValidator
GET
ValueValidator := _ValueValidator;
END_GET
END_PROPERTY

END_FUNCTION_BLOCK

// ---- Internal/CurrentNamespace.TcPOU
(*
SPDX-FileCopyrightText: © 2026 Oleksandr Tiutyk <trofimich@gmail.com>
SPDX-License-Identifier: MIT
License: https://opensource.org/license/mit
*)

(*!
<summary>Exposes the compiler-initialized namespace of Collections.</summary>
<description>
Internal metadata provider; Name borrows the extractor string and must not be modified. Do not execute this
program explicitly.
</description>
*)

{attribute 'no_explicit_call' := 'do not call this POU directly'}
PROGRAM INTERNAL CurrentNamespace
VAR
	{attribute 'hide'} 
	_NamespaceExtractor : NamespaceExtractor;
END_VAR

(*!
<summary>Borrows the compiler-initialized namespace string.</summary>
<description>
Read-only metadata backed by NamespaceExtractor; callers must not modify it.
</description>
*)
{attribute 'monitoring' := 'call'}
PROPERTY Name : REFERENCE TO STRING
GET
Name REF= _NamespaceExtractor.CurrentNamespace;
END_GET
END_PROPERTY

END_PROGRAM

// ---- Internal/NamespaceExtractor.TcPOU
(*
SPDX-FileCopyrightText: © 2026 Oleksandr Tiutyk <trofimich@gmail.com>
SPDX-License-Identifier: MIT
License: https://opensource.org/license/mit
*)

(*!
<summary>Receives compiler-initialized namespace metadata for Collections.</summary>
<description>
The exposed string remains library-owned and is read-only by contract. No allocation or runtime extraction occurs.
</description>
*)

FUNCTION_BLOCK INTERNAL NamespaceExtractor
VAR_OUTPUT
	(*!
<summary>Receives the library namespace from compiler initialization.</summary>
<description>
CurrentNamespace is populated by init_namespace and used as read-only diagnostic metadata. No runtime
extraction or allocation is performed.
</description>
*)

{attribute 'init_namespace'} 
	CurrentNamespace : STRING;	
END_VAR

END_FUNCTION_BLOCK

// ---- Dictionary/Dictionary.TcPOU
(*
SPDX-FileCopyrightText: © 2026 Oleksandr Tiutyk <trofimich@gmail.com>
SPDX-License-Identifier: MIT
License: https://opensource.org/license/mit
*)

(*!
<summary>Stores key-value entries with fixed or dynamic capacity.</summary>
<description>
CreateEnumerator allocates an independent cursor owned by its caller. The collection must remain alive while
that cursor is used. SetGeneric retains an existing matching key and replaces its value. SetGeneric preserves
disposal responsibility when the same allocation is reused; transferred caller-side owning aliases must not be
released again. Lookup uses GENERIC_VALUE equality/hashing or the borrowed keyEqualityComparer supplied once
through FB_init. Pass zero explicitly to use default key equality and hashing. Empty keys are supported unless
rejected by a validator. Raw queries create borrowed descriptors with an explicit object flag. Entries and
enumeration have no guaranteed order; positions are storage slots, not sorted ranks. Do not modify stored
descriptors through returned references. SetCopy cleans up prepared copies if preparation of the second copy
or insertion fails before ownership is accepted. Try lookup/removal operations contain exceptions without
rolling back partial effects. Generic query arguments are borrowed by default. Explicitly requested release in
Try operations is attempted even after lookup failure; caller-side owning aliases are not reset. OBJECT keys
are permitted when their descriptors refer to live Object instances. A borrowed key (IsMemoryOwner = FALSE) is
not owned or destroyed by the dictionary; its owner must keep it alive for every operation that may access the
stored key. An owned key must not be deleted or transferred to another owner through a caller-side alias.
While a key is stored, do not change data used by the active comparison rules, its equality/hash results, or
equality-relevant comparer configuration. Remove the entry before such a change, then insert it again. Queries
and callbacks must not mutate keys or reenter collection mutation. Do not use explicit query release to
dispose of a stored key or other storage still retained by the collection. An address-based identity index
must be rebuilt after address relocation; stale indices must not be used. Borrowing does not pin an object or
extend its lifetime. A copied object has its own identity; lookup using the original requires an equality
strategy under which original and copy are equal. Default OBJECT lookup delegates to
Object.Equals/GetHashCode; fields unrelated to equality/hash may change. The index caches hashes and must be
discarded and populated again after equality-relevant address relocation before further lookup. Static index
storage adds 12 bytes per capacity slot and three pointers plus the comparer reference. Dynamic entries and
the 12-byte-per-slot index share one allocation; growth temporarily retains both old and new allocations.
Expected bucket lookup is constant time plus hashing/equality costs, worst case linear; compaction and
rebuilding after removal are linear in capacity and Length. Validators are borrowed for the collection
lifetime. No internal locking is implemented. Concurrent access involving mutation requires caller
coordination; this implementation does not provide a concurrent-container guarantee. Generic lookup with
requested query release also attempts cleanup on lookup failure before propagating the captured exception;
terminal OOM takes precedence.
Instances cannot be assigned by value: copying backing pointers or disposal responsibility would create
unsafe aliases. Interface references still borrow this instance; copying an interface does not clone storage.
</description>
*)

{attribute 'no_explicit_call' := 'do not call this function block directly'}
FUNCTION_BLOCK Dictionary
VAR_GENERIC CONSTANT
 	{attribute 'hide'}
	//! <summary>Inline capacity; zero selects dynamic backing storage.</summary>
	_StaticCapacity : TOF_Core.DINT_LENGTH := 0;
END_VAR
EXTENDS TOF_Core.Object IMPLEMENTS IDictionary
VAR_INPUT
	//! <summary>Number of slots added when dynamic storage is full; must be positive when growth is required.</summary>
	DefaultDynamicAllocationElementCount : BYTE := 10;
END_VAR
VAR_STAT
	//! <summary>Class name shared by all instances of this function block.</summary>
	{attribute 'hide'}
	_ClassName : STRING := __POUNAME();
END_VAR
VAR
	{attribute 'hide'}
	_KeyValidator : TOF_Core.IGenericValueValidator;
	{attribute 'hide'}
	_ValueValidator : TOF_Core.IGenericValueValidator;
	{attribute 'hide'}
	_KeyEqualityComparer : TOF_Core.IEqualityComparer;

	{attribute 'hide'}
	_Array : POINTER TO TOF_Core.GENERIC_KEY_VALUE_PAIR;
	{attribute 'hide'}
	_StaticArray : ARRAY [0.._StaticCapacity - 1] OF TOF_Core.GENERIC_KEY_VALUE_PAIR;

	{attribute 'hide'}
	_Hashes : POINTER TO UDINT;
	{attribute 'hide'}
	_Buckets : POINTER TO DINT;
	{attribute 'hide'}
	_NextIndices : POINTER TO DINT;

	{attribute 'hide'}
	_StaticHashes : ARRAY [0.._StaticCapacity - 1] OF UDINT;
	{attribute 'hide'}
	_StaticBuckets : ARRAY [0.._StaticCapacity - 1] OF DINT;
	{attribute 'hide'}
	_StaticNextIndices : ARRAY [0.._StaticCapacity - 1] OF DINT;

	{attribute 'hide'}
	_DynamicCapacity : TOF_Core.DINT_LENGTH;
	{attribute 'hide'}
	_Length : TOF_Core.DINT_LENGTH;
END_VAR

(*!
<summary>Grows the combined entry and hash-index buffer before accepting incoming ownership.</summary>
<description>
Static collections return without allocation. A positive increment must fit DINT capacity and the UDINT
allocation-byte limit, including 12 index bytes per slot. One allocation contains entries, cached hashes,
bucket heads and links. Allocation failure preserves the old buffer, index, capacity and payload ownership and
sets terminal allocation state. Existing descriptors and hashes are copied; rebuilding links invokes no
equality/hash callbacks. Descendants cannot override this storage operation; capacity, indexing and disposal
remain governed by this collection implementation.
</description>
*)
METHOD PROTECTED FINAL AllocateMemory
VAR_INPUT
	elementCount : TOF_Core.DINT_LENGTH;
END_VAR
VAR CONSTANT
	//! <summary>Bytes per capacity slot, including descriptor storage and any hash-index arrays.</summary>
	ENTRY_ALLOCATION_SIZE : ULINT := XSIZEOF(TOF_Core.GENERIC_KEY_VALUE_PAIR) + XSIZEOF(UDINT) + 2 * XSIZEOF(DINT);
END_VAR
VAR
	newMemory : POINTER TO BYTE;
	newHashes : POINTER TO UDINT;
	newCapacity : ULINT;

END_VAR
IF NOT Dynamic THEN
	RETURN;
END_IF

IF elementCount <= TOF_Core.SignedInt32.ZERO THEN
	TOF_Core.Exceptions.ThrowArgumentOutOfRange(
		sourceNamespaceName := NamespaceName,
		sourceClassName := ClassName,
		sourcePOUName := __POUNAME(),
		sourcePosition := __POSITION(),
		argumentName := 'elementCount',
		argumentValue := elementCount
	);
END_IF

newCapacity := TO_ULINT(_DynamicCapacity) + TO_ULINT(elementCount);

IF newCapacity > TO_ULINT(TOF_Core.SignedInt32.MAX_VALUE)
	OR_ELSE newCapacity > TO_ULINT(TOF_Core.UnsignedInt32.MAX_VALUE) / ENTRY_ALLOCATION_SIZE
THEN
	TOF_Core.Exceptions.ThrowArgumentOutOfRange(
		sourceNamespaceName := NamespaceName,
		sourceClassName := ClassName,
		sourcePOUName := __POUNAME(),
		sourcePosition := __POSITION(),
		argumentName := 'capacity',
		argumentValue := newCapacity
	);
END_IF

newMemory := __NEW(BYTE, TO_UDINT(ENTRY_ALLOCATION_SIZE * newCapacity));

IF newMemory = 0 THEN
	TOF_Core.DynamicMemoryManager.RaiseAllocationFailure();
END_IF

newHashes := newMemory + TO_UDINT(XSIZEOF(TOF_Core.GENERIC_KEY_VALUE_PAIR) * newCapacity);

IF _Length > TOF_Core.SignedInt32.ZERO THEN
	Tc2_System.MEMCPY(
		destAddr := newMemory,
		srcAddr := _Array,
		n := TO_UDINT(XSIZEOF(TOF_Core.GENERIC_KEY_VALUE_PAIR) * TO_ULINT(_Length))
	);
	Tc2_System.MEMCPY(destAddr := newHashes, srcAddr := _Hashes, n := TO_UDINT(XSIZEOF(UDINT) * TO_ULINT(_Length)));
END_IF

IF _Array <> 0 THEN
	__DELETE(_Array);
END_IF

_Array := newMemory;
_Hashes := newHashes;
_Buckets := newMemory + TO_UDINT((XSIZEOF(TOF_Core.GENERIC_KEY_VALUE_PAIR) + XSIZEOF(UDINT)) * newCapacity);
_NextIndices := newMemory + TO_UDINT((XSIZEOF(TOF_Core.GENERIC_KEY_VALUE_PAIR) + XSIZEOF(UDINT) + XSIZEOF(DINT)) * newCapacity);
_DynamicCapacity := TO_DINT(newCapacity);

rebuildIndex();
END_METHOD

(*!
<summary>Reports the currently allocated number of slots.</summary>
<description>
Units are bytes for ByteList and entries for other collections. Static capacity is fixed; dynamic capacity can
change on growth or clearing. This is not a guarantee that the next allocation succeeds.
</description>
*)
{attribute 'monitoring' := 'call'}
PROPERTY FINAL Capacity : TOF_Core.DINT_LENGTH
GET
Capacity := SEL(_StaticCapacity = 0, _StaticCapacity, _DynamicCapacity);
END_GET
END_PROPERTY

(*!
<summary>Borrows the concrete collection class name without transferring storage ownership.</summary>
*)
{attribute 'monitoring' := 'call'}
PROPERTY ClassName : REFERENCE TO STRING
GET
ClassName REF= _ClassName;
END_GET
END_PROPERTY

(*!
<summary>Removes all entries and releases dynamic entry and index storage.</summary>
<description>
Owned payload cleanup is best effort. The collection is marked empty before disposal; cleanup callbacks must
not reenter mutation. Static capacity and the lifetime comparer/validators are retained. Dynamic capacity
becomes zero. Uses no allocation or equality/hash callbacks and leaves static buckets empty for reuse.
Descendants cannot override this storage operation; capacity, indexing and disposal remain governed by this
collection implementation.
</description>
*)
METHOD FINAL Clear : IDictionary
VAR
	index : DINT;
	entryCount : DINT;
END_VAR
Clear := THIS^;
entryCount := _Length;
_Length := 0;

FOR index := 0 TO entryCount - 1 DO
	_Array[index].Key.Release();
	_Array[index].Value.Release();
END_FOR

IF Dynamic THEN
	IF _Array <> 0 THEN
		__DELETE(_Array);
	END_IF

	_Array := 0;
	_Hashes := 0;
	_Buckets := 0;
	_NextIndices := 0;
	_DynamicCapacity := 0;
ELSE
	rebuildIndex();
END_IF
END_METHOD

(*!
<summary>Reports whether a matching entry exists for a borrowed generic query.</summary>
<description>
The query is borrowed by default. Explicit release requests disposal of owned query storage after lookup
completes, including a missing result. Requested release is attempted after both successful lookup and lookup
failure. Before cleanup, the original framework exception is retained and a borrowed static system exception
is cloned to preserve its code, catch point and timestamps across cleanup callbacks. The captured exception is
then propagated through ExceptionManager.Throw in the current cyclic task; native errors use the framework
SystemException representation. If capturing the system exception fails with terminal OOM, query cleanup is
still attempted and terminal OOM takes precedence. Terminal allocation state is never cleared. Release is best
effort and does not prove successful deallocation. Cleanup callbacks must not reenter collection mutation.
Release resets only the local descriptor copy; the caller must have disposal rights and must not reuse or
release owning aliases afterwards. Borrowed payload is not freed. Descendants cannot override this storage
operation; capacity, indexing and disposal remain governed by this collection implementation.
</description>
*)
METHOD FINAL ContainsGenericKey : BOOL
VAR_INPUT
	key : TOF_Core.GENERIC_VALUE;
	releaseKey : BOOL := FALSE;
END_VAR
VAR
	exceptionCode : __SYSTEM.ExceptionCode;
	caughtException : TOF_Core.IException;
END_VAR
__TRY
	ContainsGenericKey := FindKeyIndex(key := key);
__CATCH(exceptionCode)
	caughtException := TOF_Core.ExceptionManager.GetLastException(
		exceptionCode := exceptionCode,
		catchPointNamespaceName := NamespaceName,
		catchPointPOUName := __POUNAME(),
		catchPointPosition := __POSITION()
	);
__ENDTRY

IF releaseKey THEN
	IF caughtException <> 0 AND_THEN NOT caughtException.IsDynamicInstance THEN
		__TRY
			TOF_Core.DynamicMemoryManager.RaiseIfAllocationFailed();
			__QUERYINTERFACE(caughtException.Clone(), caughtException);
		__CATCH(exceptionCode)
			key.Release();

			TOF_Core.ExceptionManager.ReThrowLastException(
				exceptionCode := exceptionCode,
				catchPointNamespaceName := NamespaceName,
				catchPointPOUName := __POUNAME(),
				catchPointPosition := __POSITION()
			);
		__ENDTRY
	END_IF

	key.Release();
END_IF

IF caughtException <> 0 THEN
	TOF_Core.ExceptionManager.Throw(exception := caughtException);
END_IF
END_METHOD

(*!
<summary>Reports whether a matching raw query exists.</summary>
<description>
The raw ANY argument is borrowed without cloning or ownership transfer. keyIsObject = TRUE requires a live
Object function-block instance, not a pointer or interface variable. FALSE uses ordinary runtime type mapping.
The caller keeps the query storage alive for the call. Descendants cannot override this storage operation;
capacity, indexing and disposal remain governed by this collection implementation.
</description>
*)
//!<param name="keyIsObject">Explicitly interprets the raw argument as a live Object instance.</param>
METHOD FINAL ContainsKey : BOOL
VAR_INPUT
	key : ANY;
	keyIsObject : BOOL := FALSE;
END_VAR
VAR
	genericKey : TOF_Core.GENERIC_VALUE;
END_VAR

genericKey := TOF_Core.GenericValueFactory.FromAnyType(
		value := key,
		isObject := keyIsObject,
		memoryManagementBehavior := TOF_Core.GENERIC_MEMORY_MANAGEMENT_BEHAVIOR.STORE_ORIGINAL_REFERENCE_AND_NOT_OWNS_MEMORY
	);

ContainsKey := FindKeyIndex(key := genericKey);
END_METHOD

(*!
<summary>Creates an independent enumerator owned by the caller.</summary>
<description>
The caller must explicitly release the enumerator and keep this collection alive while using it. Allocation
failure invokes DynamicMemoryManager.RaiseAllocationFailure without a heap exception; it is terminal and is
not returned as a recoverable null result.
</description>
*)
METHOD CreateEnumerator : TOF_Core.IEnumerator
VAR
	enumerator : POINTER TO DictionaryEnumerator;
END_VAR
enumerator := __NEW(DictionaryEnumerator(dictionary := THIS^));

IF enumerator = 0 THEN
	TOF_Core.DynamicMemoryManager.RaiseAllocationFailure();
END_IF

CreateEnumerator := enumerator^;
END_METHOD

(*!
<summary>Reports whether storage can grow dynamically.</summary>
<description>
Static capacity zero selects dynamic storage. Dynamic collections can still fail to allocate.
</description>
*)
{attribute 'monitoring' := 'call'}
PROPERTY FINAL Dynamic : BOOL
GET
Dynamic := _StaticCapacity = 0;
END_GET
END_PROPERTY

(*!
<summary>Reports whether the collection has no entries.</summary>
<description>
Reflects Length; not a check of payload lifetime or memory health.
</description>
*)
{attribute 'monitoring' := 'call'}
PROPERTY FINAL Empty : BOOL
GET
Empty := _Length <= 0;
END_GET
END_PROPERTY

(*!
<summary>Releases collection payload and dynamic entry/index storage during destruction.</summary>
<description>
Calls the non-allocating Clear path without invoking equality/hash callbacks. Owned payload release is best
effort and cannot guarantee successful deallocation; cleanup callbacks must not throw or reenter mutation.
</description>
*)

METHOD FB_exit : BOOL
VAR_INPUT
	bInCopyCode : BOOL;
END_VAR
Clear();
END_METHOD

(*!
<summary>Binds validators, the lifetime equality strategy and static storage.</summary>
<description>
The key comparer is borrowed for the entire collection lifetime. Supply it explicitly; zero selects
GENERIC_VALUE default equality and hashing. Keep it alive and its equality-relevant configuration stable.
There is no subsequent comparer replacement. Initialization binds existing storage without allocating or
calling validators, comparers or other throwing paths.
</description>
*)


//!<param name="keyEqualityComparer">
//! Borrowed key equality and hash strategy; pass zero explicitly for the GENERIC_VALUE defaults.
//! </param>
METHOD FB_init : BOOL
VAR_INPUT
	bInitRetains : BOOL; // TRUE: the retain variables are initialized (reset warm / reset cold)
	bInCopyCode : BOOL; // TRUE: the instance will be copied to the copy code afterward (online change)

	keyValidator : TOF_Core.IGenericValueValidator;
	valueValidator : TOF_Core.IGenericValueValidator;
	keyEqualityComparer : TOF_Core.IEqualityComparer;
END_VAR
_KeyValidator := keyValidator;
_ValueValidator := valueValidator;
_KeyEqualityComparer := keyEqualityComparer;

IF NOT Dynamic THEN
	_Array := ADR(_StaticArray);
	_Hashes := ADR(_StaticHashes);
	_Buckets := ADR(_StaticBuckets);
	_NextIndices := ADR(_StaticNextIndices);
END_IF
END_METHOD

(*!
<summary>Finds an equal key through its hash bucket.</summary>
<description>
Borrows the descriptor and payload without changing ownership. The configured equality strategy computes the
query hash once; equal hash codes are resolved with Equals. Callback exceptions propagate before mutation. On
a miss supposedIndex is the append position. hashCode is valid after a completed lookup, including a miss. No
ordering or sorted rank is provided. Bucket heads and links encode entry index plus one; zero ends a chain.
Descendants cannot override this storage operation; capacity, indexing and disposal remain governed by this
collection implementation.
</description>
*)
METHOD PROTECTED FINAL FindKeyIndex : BOOL
VAR_INPUT
	key : TOF_Core.GENERIC_VALUE;
END_VAR
VAR_OUTPUT
	supposedIndex : DINT;
	hashCode : UDINT;
END_VAR
VAR
	entryLink : DINT;
	entryIndex : DINT;
END_VAR
FindKeyIndex := FALSE;
supposedIndex := _Length;
hashCode := key.GetHashCode(comparer := _KeyEqualityComparer);

IF _Length = TOF_Core.SignedInt32.ZERO THEN
	RETURN;
END_IF

entryLink := _Buckets[TO_DINT(hashCode MOD TO_UDINT(Capacity))];

WHILE entryLink <> TOF_Core.SignedInt32.ZERO DO
	entryIndex := entryLink - 1;

	IF _Hashes[entryIndex] = hashCode
		AND_THEN _Array[entryIndex].Key.Equals(otherValue := key, comparer := _KeyEqualityComparer)
	THEN
		supposedIndex := entryIndex;
		FindKeyIndex := TRUE;
		RETURN;
	END_IF

	entryLink := _NextIndices[entryIndex];
END_WHILE
END_METHOD

(*!
<summary>Reports whether fixed-capacity storage has no free slot.</summary>
<description>
Dynamic collections report FALSE even when Length equals Capacity. This does not guarantee available heap
memory.
</description>
*)
{attribute 'monitoring' := 'call'}
PROPERTY FINAL Full : BOOL
GET
Full := _StaticCapacity <> 0 AND_THEN _Length >= _StaticCapacity;
END_GET
END_PROPERTY

(*!
<summary>Returns the matching entry position, or a negative value when absent.</summary>
<description>
The query is borrowed by default. Explicit release requests disposal of owned query storage after lookup
completes, including a missing result. Requested release is attempted after both successful lookup and lookup
failure. Before cleanup, the original framework exception is retained and a borrowed static system exception
is cloned to preserve its code, catch point and timestamps across cleanup callbacks. The captured exception is
then propagated through ExceptionManager.Throw in the current cyclic task; native errors use the framework
SystemException representation. If capturing the system exception fails with terminal OOM, query cleanup is
still attempted and terminal OOM takes precedence. Terminal allocation state is never cleared. Release is best
effort and does not prove successful deallocation. Cleanup callbacks must not reenter collection mutation.
Release resets only the local descriptor copy; the caller must have disposal rights and must not reuse or
release owning aliases afterwards. Borrowed payload is not freed. The position is a current storage slot with
no sorted-rank guarantee; mutation may invalidate it. Descendants cannot override this storage operation;
capacity, indexing and disposal remain governed by this collection implementation.
</description>
*)
METHOD FINAL GetGenericKeyPosition : DINT
VAR_INPUT
	key : TOF_Core.GENERIC_VALUE;
	releaseKey : BOOL := FALSE;
END_VAR
VAR
	exceptionCode : __SYSTEM.ExceptionCode;
	caughtException : TOF_Core.IException;
END_VAR
__TRY
	IF NOT FindKeyIndex(key := key, supposedIndex => GetGenericKeyPosition) THEN
		GetGenericKeyPosition := -1;
	END_IF
__CATCH(exceptionCode)
	caughtException := TOF_Core.ExceptionManager.GetLastException(
		exceptionCode := exceptionCode,
		catchPointNamespaceName := NamespaceName,
		catchPointPOUName := __POUNAME(),
		catchPointPosition := __POSITION()
	);
__ENDTRY

IF releaseKey THEN
	IF caughtException <> 0 AND_THEN NOT caughtException.IsDynamicInstance THEN
		__TRY
			TOF_Core.DynamicMemoryManager.RaiseIfAllocationFailed();
			__QUERYINTERFACE(caughtException.Clone(), caughtException);
		__CATCH(exceptionCode)
			key.Release();

			TOF_Core.ExceptionManager.ReThrowLastException(
				exceptionCode := exceptionCode,
				catchPointNamespaceName := NamespaceName,
				catchPointPOUName := __POUNAME(),
				catchPointPosition := __POSITION()
			);
		__ENDTRY
	END_IF

	key.Release();
END_IF

IF caughtException <> 0 THEN
	TOF_Core.ExceptionManager.Throw(exception := caughtException);
END_IF
END_METHOD

(*!
<summary>Returns the matching storage position, or a negative value when absent.</summary>
<description>
The raw ANY argument is borrowed without cloning or ownership transfer. keyIsObject = TRUE requires a live
Object function-block instance, not a pointer or interface variable. FALSE uses ordinary runtime type mapping.
The caller keeps the query storage alive for the call. The position is a current storage slot with no
sorted-rank guarantee; mutation may invalidate it. Descendants cannot override this storage operation;
capacity, indexing and disposal remain governed by this collection implementation.
</description>
*)
//!<param name="keyIsObject">Explicitly interprets the raw argument as a live Object instance.</param>
METHOD FINAL GetKeyPosition : DINT
VAR_INPUT
	key : ANY;
	keyIsObject : BOOL := FALSE;
END_VAR
VAR
	genericKey : TOF_Core.GENERIC_VALUE;
END_VAR

genericKey := TOF_Core.GenericValueFactory.FromAnyType(
		value := key,
		isObject := keyIsObject,
		memoryManagementBehavior := TOF_Core.GENERIC_MEMORY_MANAGEMENT_BEHAVIOR.STORE_ORIGINAL_REFERENCE_AND_NOT_OWNS_MEMORY
	);

IF NOT FindKeyIndex(key := genericKey, supposedIndex => GetKeyPosition) THEN
	GetKeyPosition := -1;
END_IF
END_METHOD

(*!
<summary>Borrows the entry at a current storage position.</summary>
<description>
The index must be within Length and is not a sorted rank; otherwise an exception is raised. The returned
descriptor reference and payload remain collection-owned or borrowed from their original owner. Do not mutate
the descriptor or dispose of its payload through this view. Mutation or destruction may invalidate the
reference. Descendants cannot override this storage operation; capacity, indexing and disposal remain governed
by this collection implementation.
</description>
*)
METHOD FINAL GetKeyValuePairByIndex : REFERENCE TO TOF_Core.GENERIC_KEY_VALUE_PAIR
VAR_INPUT
	index : DINT;
END_VAR
IF index < 0 OR_ELSE index >= _Length THEN
	TOF_Core.Exceptions.ThrowArgumentOutOfRange(
		sourceNamespaceName := NamespaceName,
		sourceClassName := ClassName,
		sourcePOUName := __POUNAME(),
		sourcePosition := __POSITION(),
		argumentName := 'index',
		argumentValue := index
	);
END_IF

GetKeyValuePairByIndex REF= _Array[index];
END_METHOD

(*!
<summary>Exposes the configured key validator.</summary>
<description>
Borrowed optional reference fixed at initialization. Zero means no validator. The collection does not own or
release it.
</description>
*)
{attribute 'monitoring' := 'call'}
PROPERTY FINAL KeyValidator : TOF_Core.IGenericValueValidator
GET
KeyValidator := _KeyValidator;
END_GET
END_PROPERTY

(*!
<summary>Reports the number of stored entries.</summary>
<description>
Units are bytes for ByteList and entries for other collections. Existing positions range from zero through
Length minus one.
</description>
*)
{attribute 'monitoring' := 'call'}
PROPERTY FINAL Length : TOF_Core.DINT_LENGTH
GET
Length := _Length;
END_GET
END_PROPERTY

(*!
<summary>Provides the library namespace for diagnostics.</summary>
<description>
Borrowed read-only reference to compiler-initialized metadata; no ownership transfer.
</description>
*)
{attribute 'monitoring' := 'call'}
PROPERTY NamespaceName : REFERENCE TO STRING
GET
NamespaceName REF= CurrentNamespace.Name;
END_GET
END_PROPERTY

(*!
<summary>Rebuilds bucket chains from cached hashes after entry relocation or capacity changes.</summary>
<description>
Requires bound index storage for positive capacity and valid hashes for every live entry. Does not allocate,
access payload or invoke callbacks. This only rebuilds links; it does not recompute hashes after
equality-relevant payload or address changes.
</description>
*)
METHOD PRIVATE rebuildIndex
VAR
	index : DINT;
	bucketIndex : DINT;
END_VAR
IF Capacity = TOF_Core.SignedInt32.ZERO THEN
	RETURN;
END_IF

Tc2_System.MEMSET(destAddr := _Buckets, fillByte := 0, n := TO_UDINT(XSIZEOF(DINT) * TO_ULINT(Capacity)));

FOR index := 0 TO _Length - 1 DO
	bucketIndex := TO_DINT(_Hashes[index] MOD TO_UDINT(Capacity));
	_NextIndices[index] := _Buckets[bucketIndex];
	_Buckets[bucketIndex] := index + 1;
END_FOR
END_METHOD

(*!
<summary>Removes the entry at a current storage position.</summary>
<description>
The index must be within Length and is not a sorted rank. Entries after the removed slot are compacted and
bucket links rebuilt from cached hashes before owned payload cleanup. Index compaction and rebuilding invoke
no equality/hash callbacks and allocate no storage. Invalid indices raise an exception. Positions and borrowed
entry references may be invalidated. Payload disposal is best effort through GENERIC_VALUE.Release.
Descendants cannot override this storage operation; capacity, indexing and disposal remain governed by this
collection implementation.
</description>
*)
METHOD FINAL RemoveAt : IDictionary
VAR_INPUT
	index : DINT;
END_VAR
VAR
	removedPair : TOF_Core.GENERIC_KEY_VALUE_PAIR;
END_VAR
IF index < TOF_Core.SignedInt32.ZERO OR_ELSE index >= _Length THEN
	TOF_Core.Exceptions.ThrowArgumentOutOfRange(
		sourceNamespaceName := NamespaceName,
		sourceClassName := ClassName,
		sourcePOUName := __POUNAME(),
		sourcePosition := __POSITION(),
		argumentName := 'index',
		argumentValue := index
	);
END_IF

RemoveAt := THIS^;
removedPair := _Array[index];

IF index < _Length - 1 THEN
	Tc2_System.MEMMOVE(
		destAddr := ADR(_Array[index]),
		srcAddr := ADR(_Array[index + 1]),
		n := TO_UDINT(XSIZEOF(TOF_Core.GENERIC_KEY_VALUE_PAIR) * TO_ULINT(_Length - index - 1))
	);
	Tc2_System.MEMMOVE(
		destAddr := ADR(_Hashes[index]),
		srcAddr := ADR(_Hashes[index + 1]),
		n := TO_UDINT(XSIZEOF(UDINT) * TO_ULINT(_Length - index - 1))
	);
END_IF

_Array[_Length - 1].Key.Reset();
_Array[_Length - 1].Value.Reset();
_Length := _Length - 1;
rebuildIndex();

removedPair.Key.Release();
removedPair.Value.Release();
END_METHOD

(*!
<summary>Reports the size of this function-block instance.</summary>
<description>
Measured in bytes; includes inline storage but excludes separately allocated buffers, payload and enumerators.
</description>
*)
{attribute 'monitoring' := 'call'}
PROPERTY SelfSize : ULINT
GET
SelfSize := XSIZEOF(THIS^);
END_GET
END_PROPERTY

(*!
<summary>Creates owned copies of a key and value and stores them through SetGeneric.</summary>
<description>
Original arguments remain borrowed. Object copying requires the factory's ICloneable contract; byte copying is
shallow. Copies prepared by this call are released if copying the second argument or SetGeneric fails before
accepting ownership. Cleanup does not release the original arguments. Exceptions propagate after cleanup;
terminal allocation state is not cleared. The returned index is meaningful only on success. Descendants cannot
override this storage operation; capacity, indexing and disposal remain governed by this collection
implementation.
The original failure is captured before cleanup so nested cleanup handling cannot replace its payload.
A static native wrapper is cloned before cleanup; failure to capture still attempts prepared-copy disposal.
Terminal allocation failure takes precedence and no exception clone is allocated after its latch is set.
</description>
*)
//!<param name="key">Source key storage, borrowed during copying.</param>
//!<param name="value">Source value storage, borrowed during copying.</param>
//!<param name="keyIsObject">Explicitly interprets the key as object storage.</param>
//!<param name="valueIsObject">Explicitly interprets the value as object storage.</param>
METHOD FINAL SetCopy : IDictionary
VAR_INPUT
	key : ANY;
	value : ANY;
	keyIsObject : BOOL := FALSE;
	valueIsObject : BOOL := FALSE;
END_VAR
VAR_OUTPUT
	index : DINT;
END_VAR
VAR
	exceptionCode : __SYSTEM.ExceptionCode;
	caughtException : TOF_Core.IException;
	genericKeyValue : TOF_Core.GENERIC_VALUE;
	genericValueValue : TOF_Core.GENERIC_VALUE;
END_VAR
__TRY
	genericKeyValue := TOF_Core.GenericValueFactory.FromAnyType(
		value := key,
		isObject := keyIsObject,
		memoryManagementBehavior := TOF_Core.GENERIC_MEMORY_MANAGEMENT_BEHAVIOR.CLONE_ORIGINAL_VALUE_AND_OWNS_MEMORY
	);
	genericValueValue := TOF_Core.GenericValueFactory.FromAnyType(
		value := value,
		isObject := valueIsObject,
		memoryManagementBehavior := TOF_Core.GENERIC_MEMORY_MANAGEMENT_BEHAVIOR.CLONE_ORIGINAL_VALUE_AND_OWNS_MEMORY
	);

	SetCopy := SetGeneric(key := genericKeyValue, value := genericValueValue, index => index);
__CATCH(exceptionCode)
	caughtException := TOF_Core.ExceptionManager.GetLastException(
		exceptionCode := exceptionCode,
		catchPointNamespaceName := NamespaceName,
		catchPointPOUName := __POUNAME(),
		catchPointPosition := __POSITION()
	);
__ENDTRY

IF caughtException <> 0 THEN
	__TRY
		TOF_Core.DynamicMemoryManager.RaiseIfAllocationFailed();

		IF NOT caughtException.IsDynamicInstance THEN
			__QUERYINTERFACE(caughtException.Clone(), caughtException);
		END_IF
	__CATCH(exceptionCode)
		genericKeyValue.Release();
		genericValueValue.Release();

		TOF_Core.ExceptionManager.ReThrowLastException(
			exceptionCode := exceptionCode,
			catchPointNamespaceName := NamespaceName,
			catchPointPOUName := __POUNAME(),
			catchPointPosition := __POSITION()
		);
	__ENDTRY

	genericKeyValue.Release();
	genericValueValue.Release();

	TOF_Core.ExceptionManager.Throw(exception := caughtException);
END_IF
END_METHOD

(*!
<summary>Stores a key-value pair, retaining the existing key when a matching entry is updated.</summary>
<description>
Uses the lifetime equality/hash strategy, with no ordering guarantee. Empty descriptors are permitted unless
rejected by a validator. A successful call accepts owned arguments; borrowed payload must remain alive while
stored. Validation, lookup and growth occur before acceptance; failure before acceptance leaves incoming
ownership with the caller. An unused owned incoming key and a displaced owned value are released after the new
entry is installed, unless their allocation is retained. Reusing the same allocation preserves existing
ownership or accepts incoming ownership; it never returns ownership implicitly. When key and value alias one
allocation, the key descriptor holds the pair's disposal responsibility. Input descriptor copies are not reset
in the caller: transferred owning aliases must not be released or reused as owners. Aliases must describe the
same allocation with compatible disposal semantics; overlapping owned ranges and ownership already held by
another entry or owner are not supported. Callbacks must not mutate or reenter this collection. Cleanup is
best effort through GENERIC_VALUE.Release and does not guarantee successful deallocation. The index output is
valid only on success. Descendants cannot override this storage operation; capacity, indexing and disposal
remain governed by this collection implementation.
</description>
*)
//!<param name="key">Incoming key descriptor; owned storage is transferred on success.</param>
//!<param name="value">Incoming value descriptor; owned storage is transferred on success.</param>
METHOD FINAL SetGeneric : IDictionary
VAR_INPUT
	key : TOF_Core.GENERIC_VALUE;
	value : TOF_Core.GENERIC_VALUE;
END_VAR
VAR_OUTPUT
	index : DINT;
END_VAR
VAR

	genericKeyValuePair : TOF_Core.GENERIC_KEY_VALUE_PAIR;
	displacedValue : TOF_Core.GENERIC_VALUE;
	unusedKey : TOF_Core.GENERIC_VALUE;

	supposedIndex : DINT;
	hashCode : UDINT;
	bucketIndex : DINT;
END_VAR
IF _KeyValidator <> 0 THEN
	_KeyValidator.Validate(validatedObjectName := GetName(), valueToValidate := key);
END_IF

IF _ValueValidator <> 0 THEN
	_ValueValidator.Validate(validatedObjectName := GetName(), valueToValidate := value);
END_IF

SetGeneric := THIS^;

genericKeyValuePair.Key := key;
genericKeyValuePair.Value := value;

IF FindKeyIndex(key := genericKeyValuePair.Key, supposedIndex => supposedIndex, hashCode => hashCode) THEN
	genericKeyValuePair.Key := _Array[supposedIndex].Key;
	displacedValue := _Array[supposedIndex].Value;
	unusedKey := key;

	IF displacedValue.IsMemoryOwner THEN
		IF displacedValue.Address = genericKeyValuePair.Key.Address THEN
			IF NOT genericKeyValuePair.Key.IsMemoryOwner THEN
				genericKeyValuePair.Key := TOF_Core.GenericValueFactory.FromParts(
					genericTypeClass := genericKeyValuePair.Key.TypeClass,
					address := genericKeyValuePair.Key.Address,
					size := genericKeyValuePair.Key.Size,
					memoryManagementBehavior := TOF_Core.GENERIC_MEMORY_MANAGEMENT_BEHAVIOR.STORE_ORIGINAL_REFERENCE_AND_OWNS_MEMORY
				);
			END_IF

			displacedValue.Reset();
		ELSIF displacedValue.Address = genericKeyValuePair.Value.Address THEN
			IF NOT genericKeyValuePair.Value.IsMemoryOwner THEN
				genericKeyValuePair.Value := TOF_Core.GenericValueFactory.FromParts(
					genericTypeClass := genericKeyValuePair.Value.TypeClass,
					address := genericKeyValuePair.Value.Address,
					size := genericKeyValuePair.Value.Size,
					memoryManagementBehavior := TOF_Core.GENERIC_MEMORY_MANAGEMENT_BEHAVIOR.STORE_ORIGINAL_REFERENCE_AND_OWNS_MEMORY
				);
			END_IF

			displacedValue.Reset();
		END_IF
	END_IF

	IF unusedKey.IsMemoryOwner THEN
		IF unusedKey.Address = genericKeyValuePair.Key.Address THEN
			IF NOT genericKeyValuePair.Key.IsMemoryOwner THEN
				genericKeyValuePair.Key := TOF_Core.GenericValueFactory.FromParts(
					genericTypeClass := genericKeyValuePair.Key.TypeClass,
					address := genericKeyValuePair.Key.Address,
					size := genericKeyValuePair.Key.Size,
					memoryManagementBehavior := TOF_Core.GENERIC_MEMORY_MANAGEMENT_BEHAVIOR.STORE_ORIGINAL_REFERENCE_AND_OWNS_MEMORY
				);
			END_IF

			unusedKey.Reset();
		ELSIF unusedKey.Address = genericKeyValuePair.Value.Address THEN
			IF NOT genericKeyValuePair.Value.IsMemoryOwner THEN
				genericKeyValuePair.Value := TOF_Core.GenericValueFactory.FromParts(
					genericTypeClass := genericKeyValuePair.Value.TypeClass,
					address := genericKeyValuePair.Value.Address,
					size := genericKeyValuePair.Value.Size,
					memoryManagementBehavior := TOF_Core.GENERIC_MEMORY_MANAGEMENT_BEHAVIOR.STORE_ORIGINAL_REFERENCE_AND_OWNS_MEMORY
				);
			END_IF

			unusedKey.Reset();
		ELSIF unusedKey.Address = displacedValue.Address AND_THEN displacedValue.IsMemoryOwner THEN
			unusedKey.Reset();
		END_IF
	END_IF
ELSE
	IF _Length >= Capacity THEN
		IF Dynamic THEN
			AllocateMemory(elementCount := DefaultDynamicAllocationElementCount);
		ELSE
			TOF_Core.Exceptions.ThrowStaticCollectionFull(
				sourceNamespaceName := NamespaceName,
				sourceClassName := ClassName,
				sourcePOUName := __POUNAME(),
				sourcePosition := __POSITION(),
				collectionName := GetName(),
				capacity := TO_UDINT(Capacity)
			);
		END_IF
	END_IF
END_IF

IF genericKeyValuePair.Key.Address = genericKeyValuePair.Value.Address
	AND_THEN genericKeyValuePair.Value.IsMemoryOwner
THEN
	IF NOT genericKeyValuePair.Key.IsMemoryOwner THEN
		genericKeyValuePair.Key := TOF_Core.GenericValueFactory.FromParts(
			genericTypeClass := genericKeyValuePair.Key.TypeClass,
			address := genericKeyValuePair.Key.Address,
			size := genericKeyValuePair.Key.Size,
			memoryManagementBehavior := TOF_Core.GENERIC_MEMORY_MANAGEMENT_BEHAVIOR.STORE_ORIGINAL_REFERENCE_AND_OWNS_MEMORY
		);
	END_IF

	genericKeyValuePair.Value := TOF_Core.GenericValueFactory.FromParts(
		genericTypeClass := genericKeyValuePair.Value.TypeClass,
		address := genericKeyValuePair.Value.Address,
		size := genericKeyValuePair.Value.Size,
		memoryManagementBehavior := TOF_Core.GENERIC_MEMORY_MANAGEMENT_BEHAVIOR.STORE_ORIGINAL_REFERENCE_AND_NOT_OWNS_MEMORY
	);
END_IF

_Array[supposedIndex] := genericKeyValuePair;

IF supposedIndex = _Length THEN
	_Hashes[supposedIndex] := hashCode;
	bucketIndex := TO_DINT(hashCode MOD TO_UDINT(Capacity));
	_NextIndices[supposedIndex] := _Buckets[bucketIndex];
	_Buckets[bucketIndex] := supposedIndex + 1;
	_Length := _Length + 1;
END_IF

displacedValue.Release();
unusedKey.Release();

index := supposedIndex;
END_METHOD

(*!
<summary>Attempts to find a value by its key.</summary>
<description>
Returns TRUE when a value is found. Use the output only on TRUE; no payload is cloned. Catches exceptions
without propagating them or clearing terminal allocation state. Partial changes are not rolled back. The query
is borrowed by default. When releaseKey is explicitly TRUE, attempts to release the supplied generic argument
after lookup/removal even on failure. The caller must have disposal rights and must not reuse aliases of an
owned argument after release. A successful output is a borrowed descriptor copy; IsMemoryOwner does not
transfer disposal rights to the caller. Stored payload must not be released through the output. Descendants
cannot override this storage operation; capacity, indexing and disposal remain governed by this collection
implementation.
After nested calls and requested cleanup, a fatal allocation state forces the reported outcome to failure.
This does not roll back completed removal or reset the application-wide fatal latch.
</description>
*)
METHOD FINAL TryGetValueByGenericKey : BOOL
VAR_INPUT
	key : TOF_Core.GENERIC_VALUE;
	releaseKey : BOOL := FALSE;
END_VAR
VAR_OUTPUT
	value : TOF_Core.GENERIC_VALUE;
END_VAR
VAR
	index : DINT;
END_VAR
__TRY
	TryGetValueByGenericKey := FindKeyIndex(key := key, supposedIndex => index);

	IF TryGetValueByGenericKey THEN
		value := _Array[index].Value;
	END_IF
__CATCH
	TryGetValueByGenericKey := FALSE;
__ENDTRY

IF releaseKey THEN
	__TRY
		key.Release();
	__CATCH
		TryGetValueByGenericKey := FALSE;
	__ENDTRY
END_IF

IF TOF_Core.DynamicMemoryManager.HasAllocationFailed THEN
	TryGetValueByGenericKey := FALSE;
END_IF
END_METHOD

(*!
<summary>Attempts to find a value by its key.</summary>
<description>
Returns TRUE when a value is found. Use the output only on TRUE; no payload is cloned. Catches exceptions
without propagating them or clearing terminal allocation state. Partial changes are not rolled back. The raw
ANY argument is borrowed without cloning or ownership transfer. keyIsObject = TRUE requires a live Object
function-block instance, not a pointer or interface variable. FALSE uses ordinary runtime type mapping. The
caller keeps the query storage alive for the call. A successful output is a borrowed descriptor copy;
IsMemoryOwner does not transfer disposal rights to the caller. Stored payload must not be released through the
output. Descendants cannot override this storage operation; capacity, indexing and disposal remain governed by
this collection implementation.
After nested calls and requested cleanup, a fatal allocation state forces the reported outcome to failure.
This does not roll back completed removal or reset the application-wide fatal latch.
</description>
*)
//!<param name="keyIsObject">Explicitly interprets the raw argument as a live Object instance.</param>
METHOD FINAL TryGetValueByKey : BOOL
VAR_INPUT
	key : ANY;
	keyIsObject : BOOL := FALSE;
END_VAR
VAR_OUTPUT
	value : TOF_Core.GENERIC_VALUE;
END_VAR
VAR
	genericKey : TOF_Core.GENERIC_VALUE;
	index : DINT;
END_VAR
__TRY
	genericKey := TOF_Core.GenericValueFactory.FromAnyType(
		value := key,
		isObject := keyIsObject,
		memoryManagementBehavior := TOF_Core.GENERIC_MEMORY_MANAGEMENT_BEHAVIOR.STORE_ORIGINAL_REFERENCE_AND_NOT_OWNS_MEMORY
	);

	TryGetValueByKey := FindKeyIndex(key := genericKey, supposedIndex => index);

	IF TryGetValueByKey THEN
		value := _Array[index].Value;
	END_IF
__CATCH
	TryGetValueByKey := FALSE;
__ENDTRY

IF TOF_Core.DynamicMemoryManager.HasAllocationFailed THEN
	TryGetValueByKey := FALSE;
END_IF
END_METHOD

(*!
<summary>Attempts to remove a matching entry.</summary>
<description>
Returns the collection for chaining. removed is TRUE only after the matching entry has been removed; FALSE
means no completed removal was reported. Removal is not transactional and does not prove successful
destruction of an owned payload. Catches exceptions without propagating them or clearing terminal allocation
state. Partial changes are not rolled back. The query is borrowed by default. When releaseKey is explicitly
TRUE, attempts to release the supplied generic argument after lookup/removal even on failure. The caller must
have disposal rights and must not reuse aliases of an owned argument after release. Descendants cannot
override this storage operation; capacity, indexing and disposal remain governed by this collection
implementation.
After nested calls and requested cleanup, a fatal allocation state forces the reported outcome to failure.
This does not roll back completed removal or reset the application-wide fatal latch.
</description>
*)
METHOD FINAL TryRemoveByGenericKey : IDictionary
VAR_INPUT
	key : TOF_Core.GENERIC_VALUE;
	releaseKey : BOOL := FALSE;
END_VAR
VAR_OUTPUT
	removed : BOOL;
END_VAR
VAR
	index : DINT;
END_VAR
TryRemoveByGenericKey := THIS^;
removed := FALSE;

__TRY
	IF FindKeyIndex(key := key, supposedIndex => index) THEN
		RemoveAt(index := index);
		removed := TRUE;
	END_IF
__CATCH
	removed := FALSE;
__ENDTRY

IF releaseKey THEN
	__TRY
		key.Release();
	__CATCH
		removed := FALSE;
	__ENDTRY
END_IF

IF TOF_Core.DynamicMemoryManager.HasAllocationFailed THEN
	removed := FALSE;
END_IF
END_METHOD

(*!
<summary>Attempts to remove a matching entry.</summary>
<description>
Returns the collection for chaining. removed is TRUE only after the matching entry has been removed; FALSE
means no completed removal was reported. Removal is not transactional and does not prove successful
destruction of an owned payload. Catches exceptions without propagating them or clearing terminal allocation
state. Partial changes are not rolled back. The raw ANY argument is borrowed without cloning or ownership
transfer. keyIsObject = TRUE requires a live Object function-block instance, not a pointer or interface
variable. FALSE uses ordinary runtime type mapping. The caller keeps the query storage alive for the call.
Descendants cannot override this storage operation; capacity, indexing and disposal remain governed by this
collection implementation.
After nested calls and requested cleanup, a fatal allocation state forces the reported outcome to failure.
This does not roll back completed removal or reset the application-wide fatal latch.
</description>
*)
//!<param name="keyIsObject">Explicitly interprets the raw argument as a live Object instance.</param>
METHOD FINAL TryRemoveByKey : IDictionary
VAR_INPUT
	key : ANY;
	keyIsObject : BOOL := FALSE;
END_VAR
VAR_OUTPUT
	removed : BOOL;
END_VAR
VAR
	genericKey : TOF_Core.GENERIC_VALUE;
	index : DINT;
END_VAR
TryRemoveByKey := THIS^;
removed := FALSE;

__TRY
	genericKey := TOF_Core.GenericValueFactory.FromAnyType(
		value := key,
		isObject := keyIsObject,
		memoryManagementBehavior := TOF_Core.GENERIC_MEMORY_MANAGEMENT_BEHAVIOR.STORE_ORIGINAL_REFERENCE_AND_NOT_OWNS_MEMORY
	);

	IF FindKeyIndex(key := genericKey, supposedIndex => index) THEN
		RemoveAt(index := index);
		removed := TRUE;
	END_IF
__CATCH
	removed := FALSE;
__ENDTRY

IF TOF_Core.DynamicMemoryManager.HasAllocationFailed THEN
	removed := FALSE;
END_IF
END_METHOD

(*!
<summary>Exposes the configured value validator.</summary>
<description>
Borrowed optional reference fixed at initialization. Zero means no validator. The collection does not own or
release it.
</description>
*)
{attribute 'monitoring' := 'call'}
PROPERTY FINAL ValueValidator : TOF_Core.IGenericValueValidator
GET
ValueValidator := _ValueValidator;
END_GET
END_PROPERTY

END_FUNCTION_BLOCK

// ---- Dictionary/DictionaryEnumerator.TcPOU
(*
SPDX-FileCopyrightText: © 2026 Oleksandr Tiutyk <trofimich@gmail.com>
SPDX-License-Identifier: MIT
License: https://opensource.org/license/mit
*)

(*!
<summary>Enumerates the current storage slots of a Dictionary.</summary>
<description>
The source is borrowed and must outlive the cursor. Enumeration has no guaranteed ordering. Do not mutate the
source during traversal. Current is a borrowed view and must not be released or modified as an owning
descriptor; it is invalidated by cursor advancement/reset or source mutation. The caller owns and explicitly
releases a dynamically created cursor. MoveNext stops advancing at the end position of an unchanged source;
repeated exhausted calls return FALSE until Reset.
A null constructor source is diagnosed by traversal/current access, never by FB_init.
</description>
*)

{attribute 'no_explicit_call' := 'do not call this function block directly'}
{attribute 'enable_dynamic_creation'}
FUNCTION_BLOCK DictionaryEnumerator EXTENDS TOF_Core.Object IMPLEMENTS TOF_Core.IEnumerator
VAR_STAT
	//! <summary>Class name shared by all instances of this function block.</summary>
	{attribute 'hide'} 
	_ClassName : STRING := __POUNAME();
END_VAR
VAR
	{attribute 'hide'} 
	_Dictionary : IReadOnlyDictionary;
	{attribute 'hide'} 
	_CurrentIndex : DINT := -1;
	
	{attribute 'hide'} 
	_GenericKeyValuePair : TOF_Core.GENERIC_KEY_VALUE_PAIR;
	{attribute 'hide'} 
	_GenericValue : TOF_Core.GENERIC_VALUE;	
END_VAR

(*!
<summary>Borrows the concrete cursor class name without transferring storage ownership.</summary>
*)
{attribute 'monitoring' := 'call'}
PROPERTY ClassName : REFERENCE TO STRING
GET
ClassName REF= _ClassName;
END_GET
END_PROPERTY

(*!
<summary>Exposes a read-only borrowed view of the current entry.</summary>
<description>
Reading Current before the first successful MoveNext, after Reset or after exhaustion yields an empty
descriptor. Otherwise payload is borrowed, with no disposal rights. Do not modify or release the descriptor.
The view may change on subsequent property access, cursor movement or source mutation. The outer USER_DEFINED
value points to cursor-local GENERIC_KEY_VALUE_PAIR storage; nested descriptors borrow collection payload.
Missing source raises DataMemberNotSpecifiedException before source access or cursor advancement.
</description>
*)
{attribute 'monitoring' := 'call'}
PROPERTY FINAL Current : REFERENCE TO TOF_Core.GENERIC_VALUE
GET
requireSource();

IF _CurrentIndex >= 0 AND_THEN _CurrentIndex < _Dictionary.Length THEN
	_GenericKeyValuePair := _Dictionary.GetKeyValuePairByIndex(index := _CurrentIndex); 
	_GenericValue := TOF_Core.GenericValueFactory.FromParts(
		genericTypeClass := TOF_Core.GENERIC_TYPE_CLASS.USER_DEFINED,
		address := ADR(_GenericKeyValuePair),
		size := SIZEOF(TOF_Core.GENERIC_KEY_VALUE_PAIR),
		memoryManagementBehavior := TOF_Core.GENERIC_MEMORY_MANAGEMENT_BEHAVIOR.STORE_ORIGINAL_REFERENCE_AND_NOT_OWNS_MEMORY
	);
ELSE
	_GenericValue.Reset();
END_IF 

Current REF= _GenericValue;
END_GET
END_PROPERTY

(*!
<summary>Returns the current entry in its concrete representation.</summary>
<description>
Use only after MoveNext returns TRUE and before the next cursor or source change. No result is promised
outside a valid position. Nested descriptors borrow payload; their owner flags do not transfer disposal
rights.
Missing source raises DataMemberNotSpecifiedException before source access or cursor advancement.
</description>
*)
PROPERTY FINAL CurrentKeyValuePair : TOF_Core.GENERIC_KEY_VALUE_PAIR
GET
requireSource();

IF _CurrentIndex >= 0 AND_THEN _CurrentIndex < _Dictionary.Length THEN
	CurrentKeyValuePair := _Dictionary.GetKeyValuePairByIndex(index := _CurrentIndex); 
END_IF
END_GET
END_PROPERTY

(*!
<summary>Binds the borrowed source for enumeration.</summary>
<description>
The source must be non-null and outlive the cursor. Only the reference is assigned; no allocation, callbacks
or throwing validation are performed. A null source remains invalid configuration and is reported by
MoveNext or current-value access without throwing from initialization.
</description>
*)
METHOD FB_init : BOOL
VAR_INPUT
	bInitRetains : BOOL; // TRUE: the retain variables are initialized (reset warm / reset cold)
	bInCopyCode : BOOL;  // TRUE: the instance will be copied to the copy code afterward (online change)
	dictionary : IReadOnlyDictionary;
END_VAR
_Dictionary := dictionary;
END_METHOD

(*!
<summary>Advances the cursor to the next source position.</summary>
<description>
The source must be live, non-null and structurally unchanged during traversal. TRUE identifies a current
entry. The index advances only while below source Length and stops at the end position. Repeated exhausted
calls return FALSE without incrementing the index; reading Current yields an empty descriptor. Reset allows
traversal from the beginning again. No snapshot or mutation detection is provided.
Missing source raises DataMemberNotSpecifiedException before source access or cursor advancement.
</description>
*)
{attribute "object_name" := "MoveNext"}
METHOD FINAL MoveNext : BOOL
requireSource();

IF _CurrentIndex < _Dictionary.Length THEN
	_CurrentIndex := _CurrentIndex + 1;
END_IF

MoveNext := _CurrentIndex < _Dictionary.Length;
END_METHOD

(*!
<summary>Provides the library namespace for diagnostics.</summary>
<description>
Borrowed read-only reference to compiler-initialized metadata; no ownership transfer.
</description>
*)
{attribute 'monitoring' := 'call'}
PROPERTY NamespaceName : REFERENCE TO STRING
GET
NamespaceName REF= CurrentNamespace.Name;
END_GET
END_PROPERTY

(*!
<summary>Places the cursor before the first source entry.</summary>
<description>
The next MoveNext starts at zero. Does not modify the source or release payload; reading Current now yields an
empty descriptor. Descendants cannot override this cursor operation; advancement, reset and borrowed current
views use the same cursor state.
</description>
*)
{attribute "object_name" := "Reset"}
METHOD FINAL Reset
_CurrentIndex := -1;
END_METHOD

(*!
<summary>Reports the size of this function-block instance.</summary>
<description>
Measured in bytes; includes inline storage but excludes separately allocated buffers, payload and enumerators.
</description>
*)
{attribute 'monitoring' := 'call'}
PROPERTY SelfSize : ULINT
GET
SelfSize := XSIZEOF(THIS^);
END_GET
END_PROPERTY

(*!
<summary>Requires the configured source before traversal or current-value access.</summary>
<description>
A missing mandatory source is configuration failure, not an empty collection. Raises a framework diagnostic
outside lifecycle methods and before mutation; it does not validate arbitrary pointer lifetime.
</description>
*)
METHOD PRIVATE requireSource
IF _Dictionary = 0 THEN
	TOF_Core.Exceptions.ThrowDataMemberNotSpecified(
		sourceNamespaceName := NamespaceName,
		sourceClassName := ClassName,
		sourcePOUName := __POUNAME(),
		sourcePosition := __POSITION(),
		dataMemberName := 'dictionary'
	);
END_IF
END_METHOD

END_FUNCTION_BLOCK

// ---- Queue/QueueEnumerator.TcPOU
(*
SPDX-FileCopyrightText: © 2026 Oleksandr Tiutyk <trofimich@gmail.com>
SPDX-License-Identifier: MIT
License: https://opensource.org/license/mit
*)

(*!
<summary>Enumerates a borrowed queue using an independent cursor.</summary>
<description>
The source must be non-null, outlive the cursor and remain structurally unchanged during traversal. The caller
explicitly releases a dynamically created cursor. Current is borrowed read-only data, never an ownership
transfer. Supports both fixed-capacity and dynamic queues. MoveNext stops advancing at the end position of an
unchanged source; repeated exhausted calls return FALSE until Reset.
A null constructor source is diagnosed by traversal/current access, never by FB_init.
</description>
*)

{attribute 'no_explicit_call' := 'do not call this function block directly'}
{attribute 'enable_dynamic_creation'}
FUNCTION_BLOCK QueueEnumerator EXTENDS TOF_Core.Object IMPLEMENTS TOF_Core.IEnumerator
VAR_STAT
	//! <summary>Class name shared by all instances of this function block.</summary>
	{attribute 'hide'} 
	_ClassName : STRING := __POUNAME();
END_VAR
VAR
	{attribute 'hide'} 
	_Queue : IReadOnlyQueue;
	{attribute 'hide'} 
	_CurrentIndex : DINT := -1;
	
	{attribute 'hide'} 
	_GenericValue : TOF_Core.GENERIC_VALUE;
END_VAR

(*!
<summary>Borrows the concrete cursor class name without transferring storage ownership.</summary>
*)
{attribute 'monitoring' := 'call'}
PROPERTY ClassName : REFERENCE TO STRING
GET
ClassName REF= _ClassName;
END_GET
END_PROPERTY

(*!
<summary>Exposes a read-only borrowed view of the current entry.</summary>
<description>
Reading Current before the first successful MoveNext, after Reset or after exhaustion yields an empty
descriptor. Otherwise payload is borrowed, with no disposal rights. Do not modify or release the descriptor.
The view may change on subsequent property access, cursor movement or source mutation.
Missing source raises DataMemberNotSpecifiedException before source access or cursor advancement.
</description>
*)
{attribute 'monitoring' := 'call'}
PROPERTY FINAL Current : REFERENCE TO TOF_Core.GENERIC_VALUE
GET
requireSource();

IF _CurrentIndex >= 0 AND_THEN _CurrentIndex < _Queue.Length THEN
	_GenericValue := _Queue.GetByIndex(index := _CurrentIndex); 
ELSE
	_GenericValue.Reset();	
END_IF 

Current REF= _GenericValue;
END_GET
END_PROPERTY

(*!
<summary>Binds the borrowed source for enumeration.</summary>
<description>
The source must be non-null and outlive the cursor. Only the reference is assigned; no allocation, callbacks
or throwing validation are performed. A null source remains invalid configuration and is reported by
MoveNext or current-value access without throwing from initialization.
</description>
*)
METHOD FB_init : BOOL
VAR_INPUT
	bInitRetains : BOOL; // TRUE: the retain variables are initialized (reset warm / reset cold)
	bInCopyCode : BOOL;  // TRUE: the instance will be copied to the copy code afterward (online change)
	queue : IReadOnlyQueue;
END_VAR
_Queue := queue;
END_METHOD

(*!
<summary>Advances the cursor to the next source position.</summary>
<description>
The source must be live, non-null and structurally unchanged during traversal. TRUE identifies a current
entry. The index advances only while below source Length and stops at the end position. Repeated exhausted
calls return FALSE without incrementing the index; reading Current yields an empty descriptor. Reset allows
traversal from the beginning again. No snapshot or mutation detection is provided. Descendants cannot override
this cursor operation; advancement, reset and borrowed current views use the same cursor state.
Missing source raises DataMemberNotSpecifiedException before source access or cursor advancement.
</description>
*)
{attribute "object_name" := "MoveNext"}
METHOD FINAL MoveNext : BOOL
requireSource();

IF _CurrentIndex < _Queue.Length THEN
	_CurrentIndex := _CurrentIndex + 1;
END_IF

MoveNext := _CurrentIndex < _Queue.Length;
END_METHOD

(*!
<summary>Provides the library namespace for diagnostics.</summary>
<description>
Borrowed read-only reference to compiler-initialized metadata; no ownership transfer.
</description>
*)
{attribute 'monitoring' := 'call'}
PROPERTY NamespaceName : REFERENCE TO STRING
GET
NamespaceName REF= CurrentNamespace.Name;
END_GET
END_PROPERTY

